(* IEC 61131-3 sources: std_i2980_v2.06_cp053/Source/IMM/ieccontrol/OperationMode1, 14 files *)

(* ---- ABAlarmHandler.pu ---- *)
IMPORT_OVER_LISTFILE
 GET_ALARM_COUNT
, SET_EVENT
, tevAlarmConfirm
, tevPanelButtonRegisterData
, tevPanelButtonRegister
, tsDeviceId
, tevAlarmConfirmData

END_IMPORT

ALGORITHM_BLOCK ABAlarmHandler #DUMMY_EDIT_BLOCK

SYSTEM_VAR
 sv_iPendingAlarms : DINT;
 sv_iPendingMessages : DINT;
 di_ButtonAlarmConfirm : BOOL;
 sv_bLedAlarmConfirm_ledAttr : BYTE (* Panel LED *);
 sv_bLedAlarmConfirm : BOOL;
 sv_bHMILedAlarmConfirm_ledAttr : BYTE (* HMI LED *);
 sv_bHMILedAlarmConfirm : BOOL;
 sv_bAlarmConfirmVis : BOOL;
 sv_bButtonAlarmConfirm : BOOL;
 sv_bInitStart : BOOL;
 sv_DeviceId : tsDeviceId;
END_VAR

SYSTEM_OBJECT
 TaskVis : TASK;
 PU_Task_13 : TASK;
 evAlarmConfirm : tevAlarmConfirm;
 evPanelButtonRegister : tevPanelButtonRegister;
END_OBJECT

VAR
 mAlarmConfirmLedExists : BOOL;
 evPanelButtonRegisterData : tevPanelButtonRegisterData;
 mDIButtonAlarmConfirmLinked : BOOL;
END_VAR

VAR CONSTANT
 cButtonAlarmConfirm : DINT := 5;
END_VAR

POSTUPDATE_ALGORITHM pRegisterButtons ON PU_Task_13 WITH sv_bInitStart

#BEGIN_EDIT_BLOCK

evPanelButtonRegisterData.Button.nPanelButtonType := nPanelButtonAction;
evPanelButtonRegisterData.Button.iCompId := sv_DeviceId.CompId;
evPanelButtonRegisterData.Button.iIndexId := sv_DeviceId.IndexId;
evPanelButtonRegisterData.Button.iButtonId := cButtonAlarmConfirm;
evPanelButtonRegisterData.Button.pbActionVar1 := @sv_bButtonAlarmConfirm;
evPanelButtonRegisterData.Button.Optional.pbLedVar := @sv_bHMILedAlarmConfirm;
evPanelButtonRegisterData.Button.Optional.piLedVarAttr := @sv_bHMILedAlarmConfirm_ledAttr;
SET_EVENT(evPanelButtonRegister, evPanelButtonRegisterData);

mDIButtonAlarmConfirmLinked := IS_LINKED(di_ButtonAlarmConfirm);

;#END_EDIT_BLOCK END_ALGORITHM

PROCESS_ALGORITHM paAlarmCounter ON TaskVis AUTOSTART

VAR
 iChangeCount : DINT;
 iChangeCountOld : DINT;
END_VAR
#BEGIN_EDIT_BLOCK
(**************************************** WARNING ********************************************
 *** The KEBA Kemro K2 System including software is not intended for safety control tasks! ***
 ***                       For further information see Comment tab!                        ***
 *********************************************************************************************)

iChangeCount := GET_ALARM_MODIFICATION_COUNT();
IF iChangeCount <> iChangeCountOld THEN
   sv_iPendingAlarms := (GET_ALARM_COUNT(1)+GET_ALARM_COUNT(2)+GET_ALARM_COUNT(3));
   sv_iPendingMessages := GET_ALARM_COUNT() - sv_iPendingAlarms;
END_IF;
iChangeCountOld := iChangeCount;

;#END_EDIT_BLOCK END_ALGORITHM

POSTUPDATE_ALGORITHM pAlarmConfirmButton ON PU_Task_13 WITH di_ButtonAlarmConfirm,sv_bButtonAlarmConfirm,sv_bAlarmConfirmVis

VAR
 evAlarmConfirmData : tevAlarmConfirmData;
 bButtonAlarmConfirm : BOOL;
END_VAR
#BEGIN_EDIT_BLOCK
(**************************************** WARNING ********************************************
 *** The KEBA Kemro K2 System including software is not intended for safety control tasks! ***
 ***                       For further information see Comment tab!                        ***
 *********************************************************************************************)

bButtonAlarmConfirm := sv_bButtonAlarmConfirm;

IF mDIButtonAlarmConfirmLinked THEN
    bButtonAlarmConfirm := bButtonAlarmConfirm OR di_ButtonAlarmConfirm;
END_IF;

IF (bButtonAlarmConfirm) THEN
    //confirm button on the panel was pressed

    //confirm all alarms
    QUIT_ALARM(Name := ANY,
               SubID1 := ANY,
               SubID2 := ANY,
               SubID3 := ANY,
               SubID4 := ANY);

    //set error confirm event
    evAlarmConfirmData := nConfirmedByPanel;
    SET_EVENT(evAlarmConfirm, evAlarmConfirmData);

ELSIF sv_bAlarmConfirmVis THEN
    //alarms have been confirmed in hmi

    //set error confirm event
    evAlarmConfirmData := nConfirmedByVis;
    SET_EVENT(evAlarmConfirm, evAlarmConfirmData);
    sv_bAlarmConfirmVis := FALSE;
END_IF;

;#END_EDIT_BLOCK END_ALGORITHM

POSTUPDATE_ALGORITHM pLedControl ON PU_Task_13 WITH sv_iPendingAlarms

VAR
 bInitDone : BOOL;
END_VAR
#BEGIN_EDIT_BLOCK
(**************************************** WARNING ********************************************
 *** The KEBA Kemro K2 System including software is not intended for safety control tasks! ***
 ***                       For further information see Comment tab!                        ***
 *********************************************************************************************)

IF NOT bInitDone THEN
    sv_bHMILedAlarmConfirm_ledAttr := 16#1;
    sv_bHMILedAlarmConfirm := FALSE;

    IF (IS_LINKED(sv_bLedAlarmConfirm_ledAttr) AND IS_LINKED(sv_bLedAlarmConfirm)) THEN
        sv_bLedAlarmConfirm_ledAttr := sv_bHMILedAlarmConfirm_ledAttr;
        sv_bLedAlarmConfirm := sv_bHMILedAlarmConfirm;
        mAlarmConfirmLedExists := TRUE;
    ELSE
        mAlarmConfirmLedExists := FALSE;
    END_IF;
    bInitDone := TRUE;
END_IF;

// set the hmi button led
IF sv_iPendingAlarms = 0 THEN
    sv_bHMILedAlarmConfirm := FALSE;
ELSE
    sv_bHMILedAlarmConfirm := TRUE;
END_IF;

IF NOT mAlarmConfirmLedExists THEN
    RETURN;
END_IF;

// set the hw led
IF sv_iPendingAlarms = 0 THEN
    sv_bLedAlarmConfirm := FALSE;
ELSE
    sv_bLedAlarmConfirm := TRUE;
END_IF;

;#END_EDIT_BLOCK END_ALGORITHM

END_ALGORITHM_BLOCK

#END_OF_IEC_PART

@Puma @IecEditor 6 68 @Pou 25
@@@BEG_Comment@@@

@@@END_Comment@@@

@BEG_Contents

@BEG_Func
@RT(17)FuncTreeContainer
2
@Var @RT(15)GET_ALARM_COUNT @RT(0) @T @T @DERIVED 0 @F @RT(22)KEBA_STANDARD_FUNCTION @F
@T
@BEG_Attrib
0 @RT(0) @RT(0)
@END_Attrib
1 1 @F @F @F @F

@Var @RT(9)SET_EVENT @RT(0) @T @T @DERIVED 0 @F @RT(23)KEBA_STANDARD_PROCEDURE @F
@T
@BEG_Attrib
0 @RT(0) @RT(0)
@END_Attrib
1 1 @F @F @F @F

@END_Func

@BEG_Const
@RT(18)ConstTreeContainer
0
@END_Const

@BEG_Export

@BEG_Kind
@ALGORITHM_BLOCK @RT(14)ABAlarmHandler @STRUCTURED_TEXT
@RT(0) @RT(0) @RT(0)
@END_Kind

@BEG_Dcl
@RT(16)DclTreeContainer
19
@Var @RT(7)TaskVis @RT(0) @T @T @RENAMED 0 @T @T @DT @RT(4)TASK @RT(0) @T @T @BASIC 0 @F
@F @F
@T
@BEG_Attrib
3 @RT(0) @RT(0) @RT(0)
@END_Attrib
1 7 @F @F @F @F

@Var @RT(17)sv_iPendingAlarms @RT(0) @T @F @DT @RT(4)DINT @RT(0) @T @T @BASIC 0 @F
@F @F
@T
@BEG_Attrib
3 @RT(0) @RT(0) @RT(0)
@END_Attrib
1 8 @F @F @F @F

@Var @RT(19)sv_iPendingMessages @RT(0) @T @F @DT @RT(4)DINT @RT(0) @T @T @BASIC 0 @F
@F @F
@T
@BEG_Attrib
3 @RT(0) @RT(0) @RT(0)
@END_Attrib
1 8 @F @F @F @F

@Var @RT(21)di_ButtonAlarmConfirm @RT(0) @T @F @DT @RT(4)BOOL @RT(0) @T @T @BASIC 0 @F
@F @F
@T
@BEG_Attrib
3 @RT(0) @RT(0) @RT(0)
@END_Attrib
1 8 @F @F @F @F

@Var @RT(10)PU_Task_13 @RT(0) @T @T @RENAMED 0 @T @T @DT @RT(4)TASK @RT(0) @T @T @BASIC 0 @F
@F @F
@T
@BEG_Attrib
3 @RT(0) @RT(0) @RT(0)
@END_Attrib
1 7 @F @F @F @F

@Var @RT(27)sv_bLedAlarmConfirm_ledAttr @RT(0) @T @F @DT @RT(4)BYTE @RT(0) @T @T @BASIC 0 @F
@F @F
@T
@BEG_Attrib
3 @RT(0) @RT(9)Panel LED @RT(0)
@END_Attrib
1 8 @F @F @F @F

@Var @RT(19)sv_bLedAlarmConfirm @RT(0) @T @F @DT @RT(4)BOOL @RT(0) @T @T @BASIC 0 @F
@F @F
@T
@BEG_Attrib
3 @RT(0) @RT(0) @RT(0)
@END_Attrib
1 8 @F @F @F @F

@Var @RT(30)sv_bHMILedAlarmConfirm_ledAttr @RT(0) @T @F @DT @RT(4)BYTE @RT(0) @T @T @BASIC 0 @F
@F @F
@T
@BEG_Attrib
3 @RT(0) @RT(7)HMI LED @RT(0)
@END_Attrib
1 8 @F @F @F @F

@Var @RT(22)sv_bHMILedAlarmConfirm @RT(0) @T @F @DT @RT(4)BOOL @RT(0) @T @T @BASIC 0 @F
@F @F
@T
@BEG_Attrib
3 @RT(0) @RT(0) @RT(0)
@END_Attrib
1 8 @F @F @F @F

@Var @RT(22)mAlarmConfirmLedExists @RT(0) @T @F @DT @RT(4)BOOL @RT(0) @T @T @BASIC 0 @F
@F @F
@T
@BEG_Attrib
3 @RT(0) @RT(0) @RT(0)
@END_Attrib
1 0 @F @F @F @F

@Var @RT(19)sv_bAlarmConfirmVis @RT(0) @T @T @RENAMED 0 @T @T @DT @RT(4)BOOL @RT(0) @T @T @BASIC 0 @F
@F @F
@T
@BEG_Attrib
3 @RT(0) @RT(0) @RT(0)
@END_Attrib
1 8 @F @F @F @F

@Var @RT(22)sv_bButtonAlarmConfirm @RT(0) @T @F @DT @RT(4)BOOL @RT(0) @T @T @BASIC 0 @F
@F @F
@T
@BEG_Attrib
3 @RT(0) @RT(0) @RT(0)
@END_Attrib
1 8 @F @F @F @F

@Var @RT(14)evAlarmConfirm @RT(0) @T @T @DERIVED 0 @T @T @DT @RT(15)tevAlarmConfirm @RT(0) @T @T @UNKNOWN 0 @F
@F @F
@T
@BEG_Attrib
3 @RT(0) @RT(0) @RT(0)
@END_Attrib
1 7 @F @F @F @F

@Var @RT(25)evPanelButtonRegisterData @RT(0) @T @T @DERIVED 0 @T @T @DT @RT(26)tevPanelButtonRegisterData @RT(0) @T @T @UNKNOWN 0 @F
@F @F
@T
@BEG_Attrib
3 @RT(0) @RT(0) @RT(0)
@END_Attrib
1 0 @F @F @F @F

@Var @RT(21)evPanelButtonRegister @RT(0) @T @T @DERIVED 0 @T @T @DT @RT(22)tevPanelButtonRegister @RT(0) @T @T @UNKNOWN 0 @F
@F @F
@T
@BEG_Attrib
3 @RT(0) @RT(0) @RT(0)
@END_Attrib
1 7 @F @F @F @F

@Var @RT(13)sv_bInitStart @RT(0) @T @T @RENAMED 0 @T @T @DT @RT(4)BOOL @RT(0) @T @T @BASIC 0 @F
@F @F
@T
@BEG_Attrib
3 @RT(0) @RT(0) @RT(0)
@END_Attrib
1 8 @F @F @F @F

@Var @RT(11)sv_DeviceId @RT(0) @T @T @DERIVED 0 @T @T @DT @RT(10)tsDeviceId @RT(0) @T @T @UNKNOWN 0 @F
@F @F
@T
@BEG_Attrib
3 @RT(0) @RT(0) @RT(0)
@END_Attrib
1 8 @F @F @F @F

@Var @RT(27)mDIButtonAlarmConfirmLinked @RT(0) @T @F @DT @RT(4)BOOL @RT(0) @T @T @BASIC 0 @F
@F @F
@T
@BEG_Attrib
3 @RT(0) @RT(0) @RT(0)
@END_Attrib
1 0 @F @F @F @F

@Var @RT(19)cButtonAlarmConfirm @RT(0) @T @F @DT @RT(4)DINT @RT(0) @T @T @BASIC 0 @F
@F @F
@T
@BEG_Attrib
3 @RT(1)5 @RT(0) @RT(0)
@END_Attrib
1 15 @F @F @F @F

@END_Dcl

@END_Export

@BEG_Body

4

@BEG_Export

@BEG_Algo
@POSTUPDATE_ALGORITHM @RT(16)pRegisterButtons @STRUCTURED_TEXT
@RT(0) @RT(13)sv_bInitStart @RT(10)PU_Task_13 @F @F
@END_Algo

@BEG_Dcl
@RT(16)DclTreeContainer
0
@END_Dcl

@END_Export

@BEG_Export

@BEG_Algo
@PROCESS_ALGORITHM @RT(14)paAlarmCounter @STRUCTURED_TEXT
@RT(0) @RT(0) @RT(7)TaskVis @T @F
@END_Algo

@BEG_Dcl
@RT(16)DclTreeContainer
2
@Var @RT(12)iChangeCount @RT(0) @T @F @DT @RT(4)DINT @RT(0) @T @T @BASIC 0 @F
@F @F
@T
@BEG_Attrib
3 @RT(0) @RT(0) @RT(0)
@END_Attrib
1 0 @F @F @F @F

@Var @RT(15)iChangeCountOld @RT(0) @T @F @DT @RT(4)DINT @RT(0) @T @T @BASIC 0 @F
@F @F
@T
@BEG_Attrib
3 @RT(0) @RT(0) @RT(0)
@END_Attrib
1 0 @F @F @F @F

@END_Dcl

@END_Export

@BEG_Export

@BEG_Algo
@POSTUPDATE_ALGORITHM @RT(19)pAlarmConfirmButton @STRUCTURED_TEXT
@RT(0) @RT(64)di_ButtonAlarmConfirm,sv_bButtonAlarmConfirm,sv_bAlarmConfirmVis @RT(10)PU_Task_13 @F @F
@END_Algo

@BEG_Dcl
@RT(16)DclTreeContainer
2
@Var @RT(18)evAlarmConfirmData @RT(0) @T @T @DERIVED 0 @T @T @DT @RT(19)tevAlarmConfirmData @RT(0) @T @T @UNKNOWN 0 @F
@F @F
@T
@BEG_Attrib
3 @RT(0) @RT(0) @RT(0)
@END_Attrib
1 0 @F @F @F @F

@Var @RT(19)bButtonAlarmConfirm @RT(0) @T @F @DT @RT(4)BOOL @RT(0) @T @T @BASIC 0 @F
@F @F
@T
@BEG_Attrib
3 @RT(0) @RT(0) @RT(0)
@END_Attrib
1 0 @F @F @F @F

@END_Dcl

@END_Export

@BEG_Export

@BEG_Algo
@POSTUPDATE_ALGORITHM @RT(11)pLedControl @STRUCTURED_TEXT
@RT(0) @RT(17)sv_iPendingAlarms @RT(10)PU_Task_13 @F @F
@END_Algo

@BEG_Dcl
@RT(16)DclTreeContainer
1
@Var @RT(9)bInitDone @RT(0) @T @F @DT @RT(4)BOOL @RT(0) @T @T @BASIC 0 @F
@F @F
@T
@BEG_Attrib
3 @RT(0) @RT(0) @RT(0)
@END_Attrib
1 0 @F @F @F @F

@END_Dcl

@END_Export

@BEG_Body
@TL(12)

evPanelButtonRegisterData.Button.nPanelButtonType := nPanelButtonAction;
evPanelButtonRegisterData.Button.iCompId := sv_DeviceId.CompId;
evPanelButtonRegisterData.Button.iIndexId := sv_DeviceId.IndexId;
evPanelButtonRegisterData.Button.iButtonId := cButtonAlarmConfirm;
evPanelButtonRegisterData.Button.pbActionVar1 := @sv_bButtonAlarmConfirm;
evPanelButtonRegisterData.Button.Optional.pbLedVar := @sv_bHMILedAlarmConfirm;
evPanelButtonRegisterData.Button.Optional.piLedVarAttr := @sv_bHMILedAlarmConfirm_ledAttr;
SET_EVENT(evPanelButtonRegister, evPanelButtonRegisterData);

mDIButtonAlarmConfirmLinked := IS_LINKED(di_ButtonAlarmConfirm);

@END_Body

@@@BEG_Comment@@@
@TL(0)

@@@END_Comment@@@

@BEG_Body
@TL(15)
(**************************************** WARNING ********************************************
 *** The KEBA Kemro K2 System including software is not intended for safety control tasks! ***
 ***                       For further information see Comment tab!                        ***
 *********************************************************************************************)

iChangeCount := GET_ALARM_MODIFICATION_COUNT();
IF iChangeCount <> iChangeCountOld THEN
   sv_iPendingAlarms := (GET_ALARM_COUNT(1)+GET_ALARM_COUNT(2)+GET_ALARM_COUNT(3));
   sv_iPendingMessages := GET_ALARM_COUNT() - sv_iPendingAlarms;
END_IF;
iChangeCountOld := iChangeCount;

@END_Body

@@@BEG_Comment@@@
@TL(0)

@@@END_Comment@@@

@BEG_Body
@TL(34)
(**************************************** WARNING ********************************************
 *** The KEBA Kemro K2 System including software is not intended for safety control tasks! ***
 ***                       For further information see Comment tab!                        ***
 *********************************************************************************************)

bButtonAlarmConfirm := sv_bButtonAlarmConfirm;

IF mDIButtonAlarmConfirmLinked THEN
    bButtonAlarmConfirm := bButtonAlarmConfirm OR di_ButtonAlarmConfirm;
END_IF;

IF (bButtonAlarmConfirm) THEN
    //confirm button on the panel was pressed

    //confirm all alarms
    QUIT_ALARM(Name := ANY,
               SubID1 := ANY,
               SubID2 := ANY,
               SubID3 := ANY,
               SubID4 := ANY);

    //set error confirm event
    evAlarmConfirmData := nConfirmedByPanel;
    SET_EVENT(evAlarmConfirm, evAlarmConfirmData);

ELSIF sv_bAlarmConfirmVis THEN
    //alarms have been confirmed in hmi

    //set error confirm event
    evAlarmConfirmData := nConfirmedByVis;
    SET_EVENT(evAlarmConfirm, evAlarmConfirmData);
    sv_bAlarmConfirmVis := FALSE;
END_IF;

@END_Body

@@@BEG_Comment@@@
@TL(0)

@@@END_Comment@@@

@BEG_Body
@TL(38)
(**************************************** WARNING ********************************************
 *** The KEBA Kemro K2 System including software is not intended for safety control tasks! ***
 ***                       For further information see Comment tab!                        ***
 *********************************************************************************************)

IF NOT bInitDone THEN
    sv_bHMILedAlarmConfirm_ledAttr := 16#1;
    sv_bHMILedAlarmConfirm := FALSE;

    IF (IS_LINKED(sv_bLedAlarmConfirm_ledAttr) AND IS_LINKED(sv_bLedAlarmConfirm)) THEN
        sv_bLedAlarmConfirm_ledAttr := sv_bHMILedAlarmConfirm_ledAttr;
        sv_bLedAlarmConfirm := sv_bHMILedAlarmConfirm;
        mAlarmConfirmLedExists := TRUE;
    ELSE
        mAlarmConfirmLedExists := FALSE;
    END_IF;
    bInitDone := TRUE;
END_IF;

// set the hmi button led
IF sv_iPendingAlarms = 0 THEN
    sv_bHMILedAlarmConfirm := FALSE;
ELSE
    sv_bHMILedAlarmConfirm := TRUE;
END_IF;

IF NOT mAlarmConfirmLedExists THEN
    RETURN;
END_IF;

// set the hw led
IF sv_iPendingAlarms = 0 THEN
    sv_bLedAlarmConfirm := FALSE;
ELSE
    sv_bLedAlarmConfirm := TRUE;
END_IF;

@END_Body

@@@BEG_Comment@@@
@TL(0)

@@@END_Comment@@@
@END_Body

@END_Contents

(* ---- ABAlarmSignal.pu ---- *)
IMPORT_OVER_LISTFILE
 IS_LINKED
, ABSignalSetReset
, tevAlarmConfirm
, TON
, tevAlarmConfirmData

END_IMPORT

ALGORITHM_BLOCK ABAlarmSignal #DUMMY_EDIT_BLOCK

SYSTEM_VAR
 sv_bAutoCycleRunning : BOOL;
 do_StoppedLamp : BOOL;
 do_RunningLamp : BOOL;
 sv_bInitDone : BOOL;
 do_AlarmLamp : BOOL (* digital output for alarm lamp *);
 do_Buzzer : BOOL (* digital output for buzzer *);
 sv_iSetAlarmSignalCount : DINT (* counter how many alarms requested the alarm signal (incremented with evAlarmLampBlink event; decremented with evAlarmLampReset) *);
 sv_dBuzzerTime : TIME;
 sv_dBuzzerPulseTime : TIME;
END_VAR

SYSTEM_OBJECT
 PU_Task_7 : TASK;
 EV_Task_7 : TASK;
 TaskMid : TASK;
 evAlarmConfirm : tevAlarmConfirm;
END_OBJECT

VAR
 abSignalSetReset : ABSignalSetReset (* this AB counts the alarmevents for set and reset the alarm signals *);
 mbStopBuzzer : BOOL (* stop buzzer *);
END_VAR

POSTUPDATE_ALGORITHM pSetAlarmSignalCount ON PU_Task_7 WITH sv_bInitDone, sv_iSetAlarmSignalCount, sv_bAutoCycleRunning

VAR
 bInitDone : BOOL;
 bAlarmLampLinked : BOOL;
 bRunningLampLinked : BOOL;
 bStoppedLampLinked : BOOL;
 bBuzzerLinked : BOOL;
 iOldCount : DINT;
 iLamp : DINT;
END_VAR
#BEGIN_EDIT_BLOCK
(**************************************** WARNING ********************************************
 *** The KEBA Kemro K2 System including software is not intended for safety control tasks! ***
 ***                       For further information see Comment tab!                        ***
 *********************************************************************************************)

IF NOT bInitDone THEN
    //check if lamp or buzzer is available
    bAlarmLampLinked := IS_LINKED(do_AlarmLamp);
    bRunningLampLinked := IS_LINKED(do_RunningLamp);
    bStoppedLampLinked := IS_LINKED(do_StoppedLamp);
    bBuzzerLinked := IS_LINKED(do_Buzzer);
    bInitDone := TRUE;
END_IF;

//set or reset alarm lamp if available
IF (sv_iSetAlarmSignalCount > 0) THEN
    iLamp := 0; // alarm
ELSIF (sv_bAutoCycleRunning) THEN
    iLamp := 1; // running
ELSE
    iLamp := 2; // stopped
END_IF;

IF bAlarmLampLinked THEN
    do_AlarmLamp := iLamp = 0;
END_IF;

IF bRunningLampLinked THEN
    do_RunningLamp :=  iLamp = 1;
END_IF;

IF bStoppedLampLinked THEN
    do_StoppedLamp := iLamp = 2;
END_IF;

IF (sv_iSetAlarmSignalCount > iOldCount) AND bBuzzerLinked AND sv_dBuzzerTime > T#0ms THEN
   //start buzzer if a new alarm occured
   mbStopBuzzer := FALSE;
   START_PROCESS_ALGORITHM(paBuzzer);
ELSIF sv_iSetAlarmSignalCount = 0 THEN
   mbStopBuzzer := TRUE;
END_IF;

iOldCount := sv_iSetAlarmSignalCount;

;#END_EDIT_BLOCK END_ALGORITHM

PROCESS_ALGORITHM paBuzzer ON TaskMid

VAR
 // dActTime : TIME;
 // bUseMaxTime : BOOL (* Use max buzzer ring time, if time > 0 otherwise no use *);
 fbTimer : TON;
END_VAR

(* IecGraph-Code *)

(* init step *)
INITIAL_STEP S_Init:
END_STEP

(* steps *)
STEP S_OnTime:
AInitTimer (P);
AGenPulses (N);
END_STEP

ACTION AInitTimer: #BEGIN_EDIT_BLOCK
fbTimer(IN := FALSE, PT := sv_dBuzzerPulseTime);
do_Buzzer := TRUE;

;#END_EDIT_BLOCK END_ACTION (*AInitTimer*)
ACTION AGenPulses: #BEGIN_EDIT_BLOCK
fbTimer(IN := TRUE);
IF fbTimer.Q THEN
   do_Buzzer := NOT do_Buzzer;
   fbTimer(IN := FALSE);
END_IF;

;#END_EDIT_BLOCK END_ACTION (*AGenPulses*)
STEP S_Stop:
AStop (P);
END_STEP

ACTION AStop: #BEGIN_EDIT_BLOCK
do_Buzzer := FALSE;
STOP_PROCESS_ALGORITHM();

;#END_EDIT_BLOCK END_ACTION (*AStop*)

(* transitions *)
TRANSITION TStartBuzzer (* Trans1 *) FROM S_Init TO S_OnTime :=  #BEGIN_EDIT_BLOCK
NOT mbStopBuzzer
;#END_EDIT_BLOCK
END_TRANSITION

TRANSITION TOnTimeReached (* Trans2 *) FROM S_OnTime TO S_Stop :=  #BEGIN_EDIT_BLOCK
S_OnTime.T > sv_dBuzzerTime OR mbStopBuzzer
;#END_EDIT_BLOCK
END_TRANSITION

TRANSITION TStart (* Trans9 *) FROM S_Stop TO S_Init :=  #BEGIN_EDIT_BLOCK
TRUE
;#END_EDIT_BLOCK
END_TRANSITION

(* end IecGraph-Code *)
(* sfc-code *)
(* end sfc-code *)

END_ALGORITHM

EVENT_ALGORITHM evaAlarmConfirm ON EV_Task_7 WITH evAlarmConfirm

VAR_INPUT
 evAlarmConfirmData : tevAlarmConfirmData;
END_VAR
#BEGIN_EDIT_BLOCK
(**************************************** WARNING ********************************************
 *** The KEBA Kemro K2 System including software is not intended for safety control tasks! ***
 ***                       For further information see Comment tab!                        ***
 *********************************************************************************************)

//alarms have been confirmed by user -> stop buzzer
mbStopBuzzer := TRUE;

;#END_EDIT_BLOCK END_ALGORITHM

END_ALGORITHM_BLOCK

#END_OF_IEC_PART

@Puma @IecEditor 6 97 @Pou 25
@@@BEG_Comment@@@

@@@END_Comment@@@

@BEG_Contents

@BEG_Func
@RT(17)FuncTreeContainer
1
@Var @RT(9)IS_LINKED @RT(0) @T @T @DERIVED 0 @F @RT(22)KEBA_STANDARD_FUNCTION @F
@T
@BEG_Attrib
0 @RT(0) @RT(0)
@END_Attrib
1 1 @F @F @F @F

@END_Func

@BEG_Const
@RT(18)ConstTreeContainer
0
@END_Const

@BEG_Export

@BEG_Kind
@ALGORITHM_BLOCK @RT(13)ABAlarmSignal @STRUCTURED_TEXT
@RT(0) @RT(0) @RT(0)
@END_Kind

@BEG_Dcl
@RT(16)DclTreeContainer
15
@Var @RT(9)PU_Task_7 @RT(0) @T @T @RENAMED 0 @T @T @DT @RT(4)TASK @RT(0) @T @T @BASIC 0 @F
@F @F
@T
@BEG_Attrib
3 @RT(0) @RT(0) @RT(0)
@END_Attrib
1 7 @F @F @F @F

@Var @RT(20)sv_bAutoCycleRunning @RT(0) @T @F @DT @RT(4)BOOL @RT(0) @T @T @BASIC 0 @F
@F @F
@T
@BEG_Attrib
3 @RT(0) @RT(0) @RT(0)
@END_Attrib
1 8 @F @F @F @F

@Var @RT(14)do_StoppedLamp @RT(0) @T @F @DT @RT(4)BOOL @RT(0) @T @T @BASIC 0 @F
@F @F
@T
@BEG_Attrib
3 @RT(0) @RT(0) @RT(0)
@END_Attrib
1 8 @F @F @F @F

@Var @RT(14)do_RunningLamp @RT(0) @T @F @DT @RT(4)BOOL @RT(0) @T @T @BASIC 0 @F
@F @F
@T
@BEG_Attrib
3 @RT(0) @RT(0) @RT(0)
@END_Attrib
1 8 @F @F @F @F

@Var @RT(9)EV_Task_7 @RT(0) @T @T @RENAMED 0 @T @T @DT @RT(4)TASK @RT(0) @T @T @BASIC 0 @F
@F @F
@T
@BEG_Attrib
3 @RT(0) @RT(0) @RT(0)
@END_Attrib
1 7 @F @F @F @F

@Var @RT(12)sv_bInitDone @RT(0) @T @F @DT @RT(4)BOOL @RT(0) @T @T @BASIC 0 @F
@F @F
@T
@BEG_Attrib
3 @RT(0) @RT(0) @RT(0)
@END_Attrib
1 8 @F @F @F @F

@Var @RT(16)abSignalSetReset @RT(0) @T @T @DERIVED 0 @T @T @DT @RT(16)ABSignalSetReset @RT(0) @T @T @UNKNOWN 0 @F
@F @F
@T
@BEG_Attrib
3 @RT(0) @RT(66)this AB counts the alarmevents for set and reset the alarm signals @RT(0)
@END_Attrib
1 0 @F @F @F @F

@Var @RT(12)do_AlarmLamp @RT(0) @T @F @DT @RT(4)BOOL @RT(0) @T @T @BASIC 0 @F
@F @F
@T
@BEG_Attrib
3 @RT(0) @RT(29)digital output for alarm lamp @RT(0)
@END_Attrib
1 8 @F @F @F @F

@Var @RT(9)do_Buzzer @RT(0) @T @F @DT @RT(4)BOOL @RT(0) @T @T @BASIC 0 @F
@F @F
@T
@BEG_Attrib
3 @RT(0) @RT(25)digital output for buzzer @RT(0)
@END_Attrib
1 8 @F @F @F @F

@Var @RT(7)TaskMid @RT(0) @T @T @RENAMED 0 @T @T @DT @RT(4)TASK @RT(0) @T @T @BASIC 0 @F
@F @F
@T
@BEG_Attrib
3 @RT(0) @RT(0) @RT(0)
@END_Attrib
1 7 @F @F @F @F

@Var @RT(12)mbStopBuzzer @RT(0) @T @F @DT @RT(4)BOOL @RT(0) @T @T @BASIC 0 @F
@F @F
@T
@BEG_Attrib
3 @RT(0) @RT(11)stop buzzer @RT(0)
@END_Attrib
1 0 @F @F @F @F

@Var @RT(14)evAlarmConfirm @RT(0) @T @T @RENAMED 0 @T @T @DT @RT(15)tevAlarmConfirm @RT(0) @T @T @UNKNOWN 0 @F
@F @F
@T
@BEG_Attrib
3 @RT(0) @RT(0) @RT(0)
@END_Attrib
1 7 @F @F @F @F

@Var @RT(23)sv_iSetAlarmSignalCount @RT(0) @T @F @DT @RT(4)DINT @RT(0) @T @T @BASIC 0 @F
@F @F
@T
@BEG_Attrib
3 @RT(0) @RT(127)counter how many alarms requested the alarm signal (incremented with evAlarmLampBlink event; decremented with evAlarmLampReset) @RT(0)
@END_Attrib
1 8 @F @F @F @F

@Var @RT(14)sv_dBuzzerTime @RT(0) @T @F @DT @RT(4)TIME @RT(0) @T @T @BASIC 0 @F
@F @F
@T
@BEG_Attrib
3 @RT(0) @RT(0) @RT(0)
@END_Attrib
1 8 @F @F @F @F

@Var @RT(19)sv_dBuzzerPulseTime @RT(0) @T @F @DT @RT(4)TIME @RT(0) @T @T @BASIC 0 @F
@F @F
@T
@BEG_Attrib
3 @RT(0) @RT(0) @RT(0)
@END_Attrib
1 8 @F @F @F @F

@END_Dcl

@END_Export

@BEG_Body

3

@BEG_Export

@BEG_Algo
@POSTUPDATE_ALGORITHM @RT(20)pSetAlarmSignalCount @STRUCTURED_TEXT
@RT(0) @RT(59)sv_bInitDone, sv_iSetAlarmSignalCount, sv_bAutoCycleRunning @RT(9)PU_Task_7 @F @F
@END_Algo

@BEG_Dcl
@RT(16)DclTreeContainer
7
@Var @RT(9)bInitDone @RT(0) @T @F @DT @RT(4)BOOL @RT(0) @T @T @BASIC 0 @F
@F @F
@T
@BEG_Attrib
3 @RT(0) @RT(0) @RT(0)
@END_Attrib
1 0 @F @F @F @F

@Var @RT(16)bAlarmLampLinked @RT(0) @T @F @DT @RT(4)BOOL @RT(0) @T @T @BASIC 0 @F
@F @F
@T
@BEG_Attrib
3 @RT(0) @RT(0) @RT(0)
@END_Attrib
1 0 @F @F @F @F

@Var @RT(18)bRunningLampLinked @RT(0) @T @F @DT @RT(4)BOOL @RT(0) @T @T @BASIC 0 @F
@F @F
@T
@BEG_Attrib
3 @RT(0) @RT(0) @RT(0)
@END_Attrib
1 0 @F @F @F @F

@Var @RT(18)bStoppedLampLinked @RT(0) @T @F @DT @RT(4)BOOL @RT(0) @T @T @BASIC 0 @F
@F @F
@T
@BEG_Attrib
3 @RT(0) @RT(0) @RT(0)
@END_Attrib
1 0 @F @F @F @F

@Var @RT(13)bBuzzerLinked @RT(0) @T @F @DT @RT(4)BOOL @RT(0) @T @T @BASIC 0 @F
@F @F
@T
@BEG_Attrib
3 @RT(0) @RT(0) @RT(0)
@END_Attrib
1 0 @F @F @F @F

@Var @RT(9)iOldCount @RT(0) @T @F @DT @RT(4)DINT @RT(0) @T @T @BASIC 0 @F
@F @F
@T
@BEG_Attrib
3 @RT(0) @RT(0) @RT(0)
@END_Attrib
1 0 @F @F @F @F

@Var @RT(5)iLamp @RT(0) @T @F @DT @RT(4)DINT @RT(0) @T @T @BASIC 0 @F
@F @F
@T
@BEG_Attrib
3 @RT(0) @RT(0) @RT(0)
@END_Attrib
1 0 @F @F @F @F

@END_Dcl

@END_Export

@BEG_Export

@BEG_Algo
@PROCESS_ALGORITHM @RT(8)paBuzzer @SEQUENTIAL_FLOW_CHART
@RT(0) @RT(0) @RT(7)TaskMid @F @F
@END_Algo

@BEG_Dcl
@RT(16)DclTreeContainer
3
@Var @RT(8)dActTime @RT(0) @T @F @DT @RT(4)TIME @RT(0) @T @T @BASIC 0 @F
@F @T
@T
@BEG_Attrib
3 @RT(0) @RT(0) @RT(0)
@END_Attrib
1 0 @F @F @F @F

@Var @RT(11)bUseMaxTime @RT(0) @T @F @DT @RT(4)BOOL @RT(0) @T @T @BASIC 0 @F
@F @T
@T
@BEG_Attrib
3 @RT(0) @RT(54)Use max buzzer ring time, if time > 0 otherwise no use @RT(0)
@END_Attrib
1 0 @F @F @F @F

@Var @RT(7)fbTimer @RT(0) @T @T @DERIVED 0 @T @T @DT @RT(3)TON @RT(0) @T @T @UNKNOWN 0 @F
@F @F
@T
@BEG_Attrib
3 @RT(0) @RT(0) @RT(0)
@END_Attrib
1 0 @F @F @F @F

@END_Dcl

@END_Export

@BEG_Export

@BEG_Algo
@EVENT_ALGORITHM @RT(15)evaAlarmConfirm @STRUCTURED_TEXT
@RT(0) @RT(14)evAlarmConfirm @RT(9)EV_Task_7 @F @F
@END_Algo

@BEG_Dcl
@RT(16)DclTreeContainer
1
@Var @RT(18)evAlarmConfirmData @RT(0) @T @T @DERIVED 0 @T @T @DT @RT(19)tevAlarmConfirmData @RT(0) @T @T @UNKNOWN 0 @F
@F @F
@T
@BEG_Attrib
3 @RT(0) @RT(0) @RT(0)
@END_Attrib
1 1 @F @F @F @F

@END_Dcl

@END_Export

@BEG_Body
@TL(45)
(**************************************** WARNING ********************************************
 *** The KEBA Kemro K2 System including software is not intended for safety control tasks! ***
 ***                       For further information see Comment tab!                        ***
 *********************************************************************************************)

IF NOT bInitDone THEN
    //check if lamp or buzzer is available
    bAlarmLampLinked := IS_LINKED(do_AlarmLamp);
    bRunningLampLinked := IS_LINKED(do_RunningLamp);
    bStoppedLampLinked := IS_LINKED(do_StoppedLamp);
    bBuzzerLinked := IS_LINKED(do_Buzzer);
    bInitDone := TRUE;
END_IF;

//set or reset alarm lamp if available
IF (sv_iSetAlarmSignalCount > 0) THEN
    iLamp := 0; // alarm
ELSIF (sv_bAutoCycleRunning) THEN
    iLamp := 1; // running
ELSE
    iLamp := 2; // stopped
END_IF;

IF bAlarmLampLinked THEN
    do_AlarmLamp := iLamp = 0;
END_IF;

IF bRunningLampLinked THEN
    do_RunningLamp :=  iLamp = 1;
END_IF;

IF bStoppedLampLinked THEN
    do_StoppedLamp := iLamp = 2;
END_IF;

IF (sv_iSetAlarmSignalCount > iOldCount) AND bBuzzerLinked AND sv_dBuzzerTime > T#0ms THEN
   //start buzzer if a new alarm occured
   mbStopBuzzer := FALSE;
   START_PROCESS_ALGORITHM(paBuzzer);
ELSIF sv_iSetAlarmSignalCount = 0 THEN
   mbStopBuzzer := TRUE;
END_IF;

iOldCount := sv_iSetAlarmSignalCount;

@END_Body

@@@BEG_Comment@@@
@TL(0)

@@@END_Comment@@@

@BEG_SfcBody
10 7 12

@BEG_SfcData 2
@StepSeq @RT(4)sseq @F 1
@Loop @RT(4)loop @F 2
@StepSeq @RT(3)seq @F 5
@Step @RT(6)S_Init @F @T @F @F @RT(0) @F
@AcbCont @RT(7)unnamed @F 0

@Trans @RT(12)TStartBuzzer @F @T @F @F @T @T @TL(2)
NOT mbStopBuzzer

@RT(6)Trans1 @F
@Step @RT(8)S_OnTime @F @F @F @F @RT(0) @F
@AcbCont @RT(7)unnamed @F 2
@Acb @RT(10)AInitTimer @F @T @RT(1)P @RT(0) @F @F @T @TL(3)
fbTimer(IN := FALSE, PT := sv_dBuzzerPulseTime);
do_Buzzer := TRUE;

@F
@Acb @RT(10)AGenPulses @F @T @RT(1)N @RT(0) @F @F @T @TL(6)
fbTimer(IN := TRUE);
IF fbTimer.Q THEN
   do_Buzzer := NOT do_Buzzer;
   fbTimer(IN := FALSE);
END_IF;

@F

@Trans @RT(14)TOnTimeReached @F @T @F @F @T @T @TL(2)
S_OnTime.T > sv_dBuzzerTime OR mbStopBuzzer

@RT(6)Trans2 @F
@Step @RT(6)S_Stop @F @F @F @F @RT(0) @F
@AcbCont @RT(7)unnamed @F 1
@Acb @RT(5)AStop @F @T @RT(1)P @RT(0) @F @F @T @TL(3)
do_Buzzer := FALSE;
STOP_PROCESS_ALGORITHM();

@F

@Trans @RT(6)TStart @F @T @T @T @T @T @TL(2)
TRUE

@RT(6)Trans9 @F

@END_SfcData
@SaActions 0
@SaTrans 0
@SaExits 0
@END_SfcBody

@@@BEG_Comment@@@
@TL(0)

@@@END_Comment@@@

@BEG_Body
@TL(8)
(**************************************** WARNING ********************************************
 *** The KEBA Kemro K2 System including software is not intended for safety control tasks! ***
 ***                       For further information see Comment tab!                        ***
 *********************************************************************************************)

//alarms have been confirmed by user -> stop buzzer
mbStopBuzzer := TRUE;

@END_Body

@@@BEG_Comment@@@
@TL(0)

@@@END_Comment@@@
@END_Body

@END_Contents

(* ---- ABAlarmSignalList.pu ---- *)
IMPORT_OVER_LISTFILE
 SET_ALARM
, tsListStructAlarmSignal
, tsDeviceId
, FBDebugTrace
, tsTraceLevel
, tsElementAlarmSignal
, tsSearchDataAlarmSignal

END_IMPORT

ALGORITHM_BLOCK ABAlarmSignalList #DUMMY_EDIT_BLOCK

SYSTEM_VAR
 sv_DeviceId : tsDeviceId;
 sv_TraceLevel : tsTraceLevel;
END_VAR

SYSTEM_OBJECT
 erListOverflow : ALARM;
END_OBJECT

VAR
 mListStruct : tsListStructAlarmSignal;
 miNextFree : DINT;
 miLowBound : DINT;
 miHighBound : DINT;
 mbInit : BOOL;
 miLastFound : DINT;
 miActElement : DINT;
 fbDebugTrace : FBDebugTrace;
END_VAR

ALGORITHM aInit

#BEGIN_EDIT_BLOCK
miLowBound := GET_LOW_BOUND(mListStruct.List);
miHighBound := GET_HIGH_BOUND(mListStruct.List);
miNextFree := miLowBound;
miLastFound := miLowBound;
miActElement := miLowBound;
mbInit := TRUE;

;#END_EDIT_BLOCK END_ALGORITHM

ALGORITHM aAdd

VAR_INPUT
 Element : tsElementAlarmSignal;
END_VAR
#BEGIN_EDIT_BLOCK
IF NOT mbInit THEN RETURN;; END_IF;

IF miNextFree < miHighBound THEN

    mListStruct.List[miNextFree] := Element;
    mListStruct.Used[miNextFree] := TRUE;
    miNextFree := miNextFree + 1;
ELSE
    //error: List Full
    SET_ALARM(Name := erListOverflow,
              SubID1 := sv_DeviceId.CompId,
              SubID2 := sv_DeviceId.IndexId,
              Param1 := 'ABAlarmSignalList.aAdd');
END_IF;

;#END_EDIT_BLOCK END_ALGORITHM

ALGORITHM aAddAt

VAR_INPUT
 Element : tsElementAlarmSignal;
 iPos : DINT;
END_VAR

VAR_TEMP
 i : DINT;
END_VAR

VAR
 iStart : DINT;
 iEnd : DINT;
END_VAR
#BEGIN_EDIT_BLOCK
IF NOT mbInit THEN RETURN; END_IF;

IF miNextFree <= miHighBound THEN
    IF iPos < miHighBound AND iPos >= miLowBound THEN

        IF iPos < miNextFree THEN

            iStart := miNextFree;
            iEnd := iPos+1;
        ELSE
            i := iPos;
            iEnd := miNextFree;
        END_IF;
        miNextFree := i + 1;

        //reorganize list
        FOR i := iStart TO iEnd BY -1 DO
            mListStruct.List[i] := mListStruct.List[i-1];
            mListStruct.Used[i] := TRUE;
        END_FOR;
        //adding Element
        mListStruct.List[iPos] := Element;
        mListStruct.Used[iPos] := TRUE;
    ELSE
        //error: out of bounds
        IF sv_TraceLevel.bApplication THEN
            fbDebugTrace(sText := 'ABAlarmSignalList.aAddAt: Error: Out of ListBounds');
        END_IF;
    END_IF;
ELSE
    //error: List Full
    SET_ALARM(Name := erListOverflow,
            SubID1 := sv_DeviceId.CompId,
            SubID2 := sv_DeviceId.IndexId,
            Param1 := 'ABAlarmSignalList.aAddAt');
END_IF;

;#END_EDIT_BLOCK END_ALGORITHM

ALGORITHM aSearch

VAR_INPUT
 SearchData : tsSearchDataAlarmSignal;
END_VAR

VAR_OUTPUT
 Element : tsElementAlarmSignal;
 iPos : DINT;
 bFound : BOOL;
END_VAR

VAR_TEMP
 i : DINT;
END_VAR
#BEGIN_EDIT_BLOCK
IF NOT mbInit THEN RETURN;; END_IF;

iPos := 0;
bFound := FALSE;

FOR i := miLowBound TO miNextFree-1 DO

    IF mListStruct.List[i].SearchData = SearchData THEN

       Element := mListStruct.List[i];
       //remember foundposition for aSearchNext
       miLastFound := i;
       iPos := i;
       bFound := TRUE;
       RETURN;;
    END_IF;
END_FOR;

;#END_EDIT_BLOCK END_ALGORITHM

ALGORITHM aSearchNext

VAR_INPUT
 SearchData : tsSearchDataAlarmSignal;
END_VAR

VAR_OUTPUT
 Element : tsElementAlarmSignal;
 iPos : DINT;
 bFound : BOOL;
END_VAR

VAR_TEMP
 i : DINT;
END_VAR
#BEGIN_EDIT_BLOCK
IF NOT mbInit THEN RETURN;; END_IF;

iPos := 0;
bFound := FALSE;

FOR i := miLastFound+1 TO miNextFree-1 DO

    IF mListStruct.List[i].SearchData = SearchData THEN

       Element := mListStruct.List[i];
       //remember foundposition for then next aSearchNext
       miLastFound := i;
       iPos := i;
       bFound := TRUE;
       RETURN;;
    END_IF;
END_FOR;

;#END_EDIT_BLOCK END_ALGORITHM

ALGORITHM aRemove

VAR_INPUT
 SearchData : tsSearchDataAlarmSignal;
END_VAR

VAR_OUTPUT
 Element : tsElementAlarmSignal;
 iPos : DINT;
 bFound : BOOL;
END_VAR

VAR_TEMP
 i : DINT;
END_VAR
#BEGIN_EDIT_BLOCK
IF NOT mbInit THEN RETURN; END_IF;

iPos := 0;
bFound := FALSE;

FOR i := miLowBound TO miNextFree-1 DO

    IF mListStruct.List[i].SearchData = SearchData THEN

       iPos := i;
       bFound := TRUE;
       Element := mListStruct.List[i];
       //reorganize list
       FOR i := iPos TO miNextFree-1 DO
           mListStruct.List[i] := mListStruct.List[i+1];
       END_FOR;
       mListStruct.Used[miNextFree-1] := FALSE;
       miNextFree := miNextFree - 1;
       RETURN;
    END_IF;
END_FOR;

;#END_EDIT_BLOCK END_ALGORITHM

ALGORITHM aRemoveAt

VAR_INPUT
 iPos : DINT;
END_VAR

VAR_OUTPUT
 Element : tsElementAlarmSignal;
END_VAR

VAR_TEMP
 i : DINT;
END_VAR
#BEGIN_EDIT_BLOCK
IF NOT mbInit THEN RETURN; END_IF;

IF iPos <= miHighBound AND iPos >= miLowBound THEN

    Element:= mListStruct.List[iPos];
    miActElement := iPos;

    //reorganize list
    FOR i := iPos TO miNextFree-1 DO
        mListStruct.List[i] := mListStruct.List[i+1];
    END_FOR;
    mListStruct.Used[miNextFree-1] := FALSE;

    miNextFree := miNextFree - 1;
ELSE
    //error: out of bounds
    IF sv_TraceLevel.bApplication THEN
        fbDebugTrace(sText := 'ABAlarmSignalList.aRemoveAt: Error: Out of ListBounds');
    END_IF;
END_IF;

;#END_EDIT_BLOCK END_ALGORITHM

ALGORITHM aRemoveAll

VAR_TEMP
 i : DINT;
END_VAR
#BEGIN_EDIT_BLOCK
IF NOT mbInit THEN RETURN; END_IF;
FOR i := miNextFree-1 TO miLowBound DO
    //clearing the whole list
    mListStruct.Used[i] := FALSE;
END_FOR;
miNextFree := miLowBound;

;#END_EDIT_BLOCK END_ALGORITHM

ALGORITHM aElementAt

VAR_OUTPUT
 Element : tsElementAlarmSignal;
END_VAR

VAR_INPUT
 iPos : DINT;
END_VAR
#BEGIN_EDIT_BLOCK
IF NOT mbInit THEN RETURN; END_IF;

IF iPos <= miHighBound AND iPos >= miLowBound THEN

    Element := mListStruct.List[iPos];
    miActElement := iPos;
ELSE
    //error: out of bounds
    IF sv_TraceLevel.bApplication THEN
        fbDebugTrace(sText := 'ABAlarmSignalList.aElementAt: Error: Out of ListBounds');
    END_IF;
END_IF;

;#END_EDIT_BLOCK END_ALGORITHM

ALGORITHM aModifyAt

VAR_INPUT
 iPos : DINT;
END_VAR

VAR_IN_OUT
 Element : tsElementAlarmSignal;
END_VAR
#BEGIN_EDIT_BLOCK
IF NOT mbInit THEN RETURN; END_IF;

IF iPos <= miHighBound AND iPos >= miLowBound THEN

     mListStruct.List[iPos] := Element;
     miActElement := iPos;
ELSE
    //error: out of bounds
    IF sv_TraceLevel.bApplication THEN
        fbDebugTrace(sText := 'ABAlarmSignalList.aModifyAt: Error: Out of ListBounds');
    END_IF;
END_IF;

;#END_EDIT_BLOCK END_ALGORITHM

// ALGORITHM aGetSize

// #BEGIN_EDIT_BLOCK
// IF NOT mbInit THEN RETURN; END_IF;
// //returns the size of the list
// iSize := miHighBound - miLowBound;

// ;#END_EDIT_BLOCK END_ALGORITHM

// ALGORITHM aGetElementsCount

// VAR_OUTPUT
 // iUsed : DINT;
// END_VAR
// #BEGIN_EDIT_BLOCK
// IF NOT mbInit THEN RETURN; END_IF;
//
// iUsed := miNextFree - miLowBound;

// ;#END_EDIT_BLOCK END_ALGORITHM

FUNCTION aGetSize : DINT
 #DUMMY_EDIT_BLOCK
#BEGIN_EDIT_BLOCK
IF NOT mbInit THEN RETURN; END_IF;
//returns the size of the list
aGetSize := miHighBound - miLowBound;

;#END_EDIT_BLOCK END_FUNCTION

FUNCTION aGetElementCount : DINT
 #DUMMY_EDIT_BLOCK
#BEGIN_EDIT_BLOCK
IF NOT mbInit THEN RETURN; END_IF;

aGetElementCount:= miNextFree - miLowBound;

;#END_EDIT_BLOCK END_FUNCTION

ALGORITHM aFirstElement

VAR_OUTPUT
 Element : tsElementAlarmSignal;
END_VAR
#BEGIN_EDIT_BLOCK
IF NOT mbInit THEN RETURN; END_IF;

miActElement := miLowBound;
Element := mListStruct.List[miLowBound];

;#END_EDIT_BLOCK END_ALGORITHM

ALGORITHM aNextElement

VAR_OUTPUT
 Element : tsElementAlarmSignal;
 iPos : DINT;
END_VAR
#BEGIN_EDIT_BLOCK
IF NOT mbInit THEN RETURN; END_IF;

IF miActElement < miHighBound THEN

    miActElement := miActElement + 1;
    iPos := miActElement;
    Element := mListStruct.List[miActElement];
END_IF;

;#END_EDIT_BLOCK END_ALGORITHM

ALGORITHM aLastElement

VAR_OUTPUT
 Element : tsElementAlarmSignal;
END_VAR
#BEGIN_EDIT_BLOCK
IF NOT mbInit THEN RETURN; END_IF;

miActElement := miNextFree - 1;
Element := mListStruct.List[miActElement];

;#END_EDIT_BLOCK END_ALGORITHM

ALGORITHM aPrevElement

VAR_OUTPUT
 Element : tsElementAlarmSignal;
 iPos : DINT;
END_VAR
#BEGIN_EDIT_BLOCK
IF NOT mbInit THEN RETURN; END_IF;

IF miActElement > miLowBound THEN

    miActElement := miActElement - 1;
    iPos := miActElement;
    Element := mListStruct.List[miActElement];
END_IF;

;#END_EDIT_BLOCK END_ALGORITHM

ALGORITHM aImport

VAR_INPUT
 ListStruct : tsListStructAlarmSignal;
END_VAR

VAR_TEMP
 i : DINT;
END_VAR
#BEGIN_EDIT_BLOCK
IF NOT mbInit THEN RETURN; END_IF;

miLastFound := miLowBound;
miActElement := miLowBound;
miNextFree := miLowBound;
mListStruct :=  ListStruct;

//cheching used elements
FOR i := miLowBound TO miHighBound DO

   IF NOT mListStruct.Used[i] THEN
        miNextFree := i;
        RETURN;
   END_IF;
END_FOR;

;#END_EDIT_BLOCK END_ALGORITHM

ALGORITHM aExport

VAR_OUTPUT
 ListStruct : tsListStructAlarmSignal;
END_VAR
#BEGIN_EDIT_BLOCK
IF NOT mbInit THEN RETURN; END_IF;

ListStruct := mListStruct;

;#END_EDIT_BLOCK END_ALGORITHM

END_ALGORITHM_BLOCK

#END_OF_IEC_PART

@Puma @IecEditor 6 68 @Pou 25
@@@BEG_Comment@@@

@@@END_Comment@@@

@BEG_Contents

@BEG_Func
@RT(17)FuncTreeContainer
1
@Var @RT(9)SET_ALARM @RT(0) @T @T @DERIVED 0 @F @RT(23)KEBA_STANDARD_PROCEDURE @F
@T
@BEG_Attrib
0 @RT(0) @RT(0)
@END_Attrib
1 1 @F @F @F @F

@END_Func

@BEG_Const
@RT(18)ConstTreeContainer
0
@END_Const

@BEG_Export

@BEG_Kind
@ALGORITHM_BLOCK @RT(17)ABAlarmSignalList @STRUCTURED_TEXT
@RT(0) @RT(0) @RT(0)
@END_Kind

@BEG_Dcl
@RT(16)DclTreeContainer
11
@Var @RT(14)erListOverflow @RT(0) @T @F @DT @RT(5)ALARM @RT(0) @T @T @BASIC 0 @F
@F @F
@T
@BEG_Attrib
3 @RT(0) @RT(0) @RT(0)
@END_Attrib
1 7 @F @F @F @F

@Var @RT(11)mListStruct @RT(0) @T @T @DERIVED 0 @T @T @DT @RT(23)tsListStructAlarmSignal @RT(0) @T @T @UNKNOWN 0 @F
@F @F
@T
@BEG_Attrib
3 @RT(0) @RT(0) @RT(0)
@END_Attrib
1 0 @F @F @F @F

@Var @RT(10)miNextFree @RT(0) @T @F @DT @RT(4)DINT @RT(0) @T @T @BASIC 0 @F
@F @F
@T
@BEG_Attrib
3 @RT(0) @RT(0) @RT(0)
@END_Attrib
1 0 @F @F @F @F

@Var @RT(10)miLowBound @RT(0) @T @F @DT @RT(4)DINT @RT(0) @T @T @BASIC 0 @F
@F @F
@T
@BEG_Attrib
3 @RT(0) @RT(0) @RT(0)
@END_Attrib
1 0 @F @F @F @F

@Var @RT(11)miHighBound @RT(0) @T @F @DT @RT(4)DINT @RT(0) @T @T @BASIC 0 @F
@F @F
@T
@BEG_Attrib
3 @RT(0) @RT(0) @RT(0)
@END_Attrib
1 0 @F @F @F @F

@Var @RT(6)mbInit @RT(0) @T @F @DT @RT(4)BOOL @RT(0) @T @T @BASIC 0 @F
@F @F
@T
@BEG_Attrib
3 @RT(0) @RT(0) @RT(0)
@END_Attrib
1 0 @F @F @F @F

@Var @RT(11)miLastFound @RT(0) @T @F @DT @RT(4)DINT @RT(0) @T @T @BASIC 0 @F
@F @F
@T
@BEG_Attrib
3 @RT(0) @RT(0) @RT(0)
@END_Attrib
1 0 @F @F @F @F

@Var @RT(12)miActElement @RT(0) @T @F @DT @RT(4)DINT @RT(0) @T @T @BASIC 0 @F
@F @F
@T
@BEG_Attrib
3 @RT(0) @RT(0) @RT(0)
@END_Attrib
1 0 @F @F @F @F

@Var @RT(11)sv_DeviceId @RT(0) @T @T @DERIVED 0 @T @T @DT @RT(10)tsDeviceId @RT(0) @T @T @UNKNOWN 0 @F
@F @F
@T
@BEG_Attrib
3 @RT(0) @RT(0) @RT(0)
@END_Attrib
1 8 @F @F @F @F

@Var @RT(12)fbDebugTrace @RT(0) @T @T @DERIVED 0 @T @T @DT @RT(12)FBDebugTrace @RT(0) @T @T @UNKNOWN 0 @F
@F @F
@T
@BEG_Attrib
3 @RT(0) @RT(0) @RT(0)
@END_Attrib
1 0 @F @F @F @F

@Var @RT(13)sv_TraceLevel @RT(0) @T @T @DERIVED 0 @T @T @DT @RT(12)tsTraceLevel @RT(0) @T @T @UNKNOWN 0 @F
@F @F
@T
@BEG_Attrib
3 @RT(0) @RT(0) @RT(0)
@END_Attrib
1 8 @F @F @F @F

@END_Dcl

@END_Export

@BEG_Body

20

@BEG_Export

@BEG_Algo
@ALGORITHM @RT(5)aInit @STRUCTURED_TEXT
@RT(0) @RT(0) @RT(0) @F @F
@END_Algo

@BEG_Dcl
@RT(16)DclTreeContainer
0
@END_Dcl

@END_Export

@BEG_Export

@BEG_Algo
@ALGORITHM @RT(4)aAdd @STRUCTURED_TEXT
@RT(0) @RT(0) @RT(0) @F @F
@END_Algo

@BEG_Dcl
@RT(16)DclTreeContainer
1
@Var @RT(7)Element @RT(0) @T @T @DERIVED 0 @T @T @DT @RT(20)tsElementAlarmSignal @RT(0) @T @T @UNKNOWN 0 @F
@F @F
@T
@BEG_Attrib
3 @RT(0) @RT(0) @RT(0)
@END_Attrib
1 1 @F @F @F @F

@END_Dcl

@END_Export

@BEG_Export

@BEG_Algo
@ALGORITHM @RT(6)aAddAt @STRUCTURED_TEXT
@RT(0) @RT(0) @RT(0) @F @F
@END_Algo

@BEG_Dcl
@RT(16)DclTreeContainer
5
@Var @RT(7)Element @RT(0) @T @T @DERIVED 0 @T @T @DT @RT(20)tsElementAlarmSignal @RT(0) @T @T @UNKNOWN 0 @F
@F @F
@T
@BEG_Attrib
3 @RT(0) @RT(0) @RT(0)
@END_Attrib
1 1 @F @F @F @F

@Var @RT(4)iPos @RT(0) @T @F @DT @RT(4)DINT @RT(0) @T @T @BASIC 0 @F
@F @F
@T
@BEG_Attrib
3 @RT(0) @RT(0) @RT(0)
@END_Attrib
1 1 @F @F @F @F

@Var @RT(1)i @RT(0) @T @F @DT @RT(4)DINT @RT(0) @T @T @BASIC 0 @F
@F @F
@T
@BEG_Attrib
3 @RT(0) @RT(0) @RT(0)
@END_Attrib
1 4 @F @F @F @F

@Var @RT(6)iStart @RT(0) @T @F @DT @RT(4)DINT @RT(0) @T @T @BASIC 0 @F
@F @F
@T
@BEG_Attrib
3 @RT(0) @RT(0) @RT(0)
@END_Attrib
1 0 @F @F @F @F

@Var @RT(4)iEnd @RT(0) @T @F @DT @RT(4)DINT @RT(0) @T @T @BASIC 0 @F
@F @F
@T
@BEG_Attrib
3 @RT(0) @RT(0) @RT(0)
@END_Attrib
1 0 @F @F @F @F

@END_Dcl

@END_Export

@BEG_Export

@BEG_Algo
@ALGORITHM @RT(7)aSearch @STRUCTURED_TEXT
@RT(0) @RT(0) @RT(0) @F @F
@END_Algo

@BEG_Dcl
@RT(16)DclTreeContainer
5
@Var @RT(10)SearchData @RT(0) @T @T @DERIVED 0 @T @T @DT @RT(23)tsSearchDataAlarmSignal @RT(0) @T @T @UNKNOWN 0 @F
@F @F
@T
@BEG_Attrib
3 @RT(0) @RT(0) @RT(0)
@END_Attrib
1 1 @F @F @F @F

@Var @RT(7)Element @RT(0) @T @T @DERIVED 0 @T @T @DT @RT(20)tsElementAlarmSignal @RT(0) @T @T @UNKNOWN 0 @F
@F @F
@T
@BEG_Attrib
3 @RT(0) @RT(0) @RT(0)
@END_Attrib
1 3 @F @F @F @F

@Var @RT(4)iPos @RT(0) @T @F @DT @RT(4)DINT @RT(0) @T @T @BASIC 0 @F
@F @F
@T
@BEG_Attrib
3 @RT(0) @RT(0) @RT(0)
@END_Attrib
1 3 @F @F @F @F

@Var @RT(6)bFound @RT(0) @T @F @DT @RT(4)BOOL @RT(0) @T @T @BASIC 0 @F
@F @F
@T
@BEG_Attrib
3 @RT(0) @RT(0) @RT(0)
@END_Attrib
1 3 @F @F @F @F

@Var @RT(1)i @RT(0) @T @F @DT @RT(4)DINT @RT(0) @T @T @BASIC 0 @F
@F @F
@T
@BEG_Attrib
3 @RT(0) @RT(0) @RT(0)
@END_Attrib
1 4 @F @F @F @F

@END_Dcl

@END_Export

@BEG_Export

@BEG_Algo
@ALGORITHM @RT(11)aSearchNext @STRUCTURED_TEXT
@RT(0) @RT(0) @RT(0) @F @F
@END_Algo

@BEG_Dcl
@RT(16)DclTreeContainer
5
@Var @RT(10)SearchData @RT(0) @T @T @DERIVED 0 @T @T @DT @RT(23)tsSearchDataAlarmSignal @RT(0) @T @T @UNKNOWN 0 @F
@F @F
@T
@BEG_Attrib
3 @RT(0) @RT(0) @RT(0)
@END_Attrib
1 1 @F @F @F @F

@Var @RT(7)Element @RT(0) @T @T @DERIVED 0 @T @T @DT @RT(20)tsElementAlarmSignal @RT(0) @T @T @UNKNOWN 0 @F
@F @F
@T
@BEG_Attrib
3 @RT(0) @RT(0) @RT(0)
@END_Attrib
1 3 @F @F @F @F

@Var @RT(4)iPos @RT(0) @T @F @DT @RT(4)DINT @RT(0) @T @T @BASIC 0 @F
@F @F
@T
@BEG_Attrib
3 @RT(0) @RT(0) @RT(0)
@END_Attrib
1 3 @F @F @F @F

@Var @RT(6)bFound @RT(0) @T @F @DT @RT(4)BOOL @RT(0) @T @T @BASIC 0 @F
@F @F
@T
@BEG_Attrib
3 @RT(0) @RT(0) @RT(0)
@END_Attrib
1 3 @F @F @F @F

@Var @RT(1)i @RT(0) @T @F @DT @RT(4)DINT @RT(0) @T @T @BASIC 0 @F
@F @F
@T
@BEG_Attrib
3 @RT(0) @RT(0) @RT(0)
@END_Attrib
1 4 @F @F @F @F

@END_Dcl

@END_Export

@BEG_Export

@BEG_Algo
@ALGORITHM @RT(7)aRemove @STRUCTURED_TEXT
@RT(0) @RT(0) @RT(0) @F @F
@END_Algo

@BEG_Dcl
@RT(16)DclTreeContainer
5
@Var @RT(10)SearchData @RT(0) @T @T @DERIVED 0 @T @T @DT @RT(23)tsSearchDataAlarmSignal @RT(0) @T @T @UNKNOWN 0 @F
@F @F
@T
@BEG_Attrib
3 @RT(0) @RT(0) @RT(0)
@END_Attrib
1 1 @F @F @F @F

@Var @RT(7)Element @RT(0) @T @T @DERIVED 0 @T @T @DT @RT(20)tsElementAlarmSignal @RT(0) @T @T @UNKNOWN 0 @F
@F @F
@T
@BEG_Attrib
3 @RT(0) @RT(0) @RT(0)
@END_Attrib
1 3 @F @F @F @F

@Var @RT(4)iPos @RT(0) @T @F @DT @RT(4)DINT @RT(0) @T @T @BASIC 0 @F
@F @F
@T
@BEG_Attrib
3 @RT(0) @RT(0) @RT(0)
@END_Attrib
1 3 @F @F @F @F

@Var @RT(6)bFound @RT(0) @T @F @DT @RT(4)BOOL @RT(0) @T @T @BASIC 0 @F
@F @F
@T
@BEG_Attrib
3 @RT(0) @RT(0) @RT(0)
@END_Attrib
1 3 @F @F @F @F

@Var @RT(1)i @RT(0) @T @F @DT @RT(4)DINT @RT(0) @T @T @BASIC 0 @F
@F @F
@T
@BEG_Attrib
3 @RT(0) @RT(0) @RT(0)
@END_Attrib
1 4 @F @F @F @F

@END_Dcl

@END_Export

@BEG_Export

@BEG_Algo
@ALGORITHM @RT(9)aRemoveAt @STRUCTURED_TEXT
@RT(0) @RT(0) @RT(0) @F @F
@END_Algo

@BEG_Dcl
@RT(16)DclTreeContainer
3
@Var @RT(4)iPos @RT(0) @T @F @DT @RT(4)DINT @RT(0) @T @T @BASIC 0 @F
@F @F
@T
@BEG_Attrib
3 @RT(0) @RT(0) @RT(0)
@END_Attrib
1 1 @F @F @F @F

@Var @RT(7)Element @RT(0) @T @T @DERIVED 0 @T @T @DT @RT(20)tsElementAlarmSignal @RT(0) @T @T @UNKNOWN 0 @F
@F @F
@T
@BEG_Attrib
3 @RT(0) @RT(0) @RT(0)
@END_Attrib
1 3 @F @F @F @F

@Var @RT(1)i @RT(0) @T @F @DT @RT(4)DINT @RT(0) @T @T @BASIC 0 @F
@F @F
@T
@BEG_Attrib
3 @RT(0) @RT(0) @RT(0)
@END_Attrib
1 4 @F @F @F @F

@END_Dcl

@END_Export

@BEG_Export

@BEG_Algo
@ALGORITHM @RT(10)aRemoveAll @STRUCTURED_TEXT
@RT(0) @RT(0) @RT(0) @F @F
@END_Algo

@BEG_Dcl
@RT(16)DclTreeContainer
1
@Var @RT(1)i @RT(0) @T @F @DT @RT(4)DINT @RT(0) @T @T @BASIC 0 @F
@F @F
@T
@BEG_Attrib
3 @RT(0) @RT(0) @RT(0)
@END_Attrib
1 4 @F @F @F @F

@END_Dcl

@END_Export

@BEG_Export

@BEG_Algo
@ALGORITHM @RT(10)aElementAt @STRUCTURED_TEXT
@RT(0) @RT(0) @RT(0) @F @F
@END_Algo

@BEG_Dcl
@RT(16)DclTreeContainer
2
@Var @RT(7)Element @RT(0) @T @T @DERIVED 0 @T @T @DT @RT(20)tsElementAlarmSignal @RT(0) @T @T @UNKNOWN 0 @F
@F @F
@T
@BEG_Attrib
3 @RT(0) @RT(0) @RT(0)
@END_Attrib
1 3 @F @F @F @F

@Var @RT(4)iPos @RT(0) @T @F @DT @RT(4)DINT @RT(0) @T @T @BASIC 0 @F
@F @F
@T
@BEG_Attrib
3 @RT(0) @RT(0) @RT(0)
@END_Attrib
1 1 @F @F @F @F

@END_Dcl

@END_Export

@BEG_Export

@BEG_Algo
@ALGORITHM @RT(9)aModifyAt @STRUCTURED_TEXT
@RT(0) @RT(0) @RT(0) @F @F
@END_Algo

@BEG_Dcl
@RT(16)DclTreeContainer
2
@Var @RT(4)iPos @RT(0) @T @F @DT @RT(4)DINT @RT(0) @T @T @BASIC 0 @F
@F @F
@T
@BEG_Attrib
3 @RT(0) @RT(0) @RT(0)
@END_Attrib
1 1 @F @F @F @F

@Var @RT(7)Element @RT(0) @T @T @DERIVED 0 @T @T @DT @RT(20)tsElementAlarmSignal @RT(0) @T @T @UNKNOWN 0 @F
@F @F
@T
@BEG_Attrib
3 @RT(0) @RT(0) @RT(0)
@END_Attrib
1 2 @F @F @F @F

@END_Dcl

@END_Export

@BEG_Export

@BEG_Algo
@ALGORITHM @RT(8)aGetSize @STRUCTURED_TEXT
@RT(0) @RT(0) @RT(0) @F @T
@END_Algo

@BEG_Dcl
@RT(16)DclTreeContainer
0
@END_Dcl

@END_Export

@BEG_Export

@BEG_Algo
@ALGORITHM @RT(17)aGetElementsCount @STRUCTURED_TEXT
@RT(0) @RT(0) @RT(0) @F @T
@END_Algo

@BEG_Dcl
@RT(16)DclTreeContainer
1
@Var @RT(5)iUsed @RT(0) @T @F @DT @RT(4)DINT @RT(0) @T @T @BASIC 0 @F
@F @F
@T
@BEG_Attrib
3 @RT(0) @RT(0) @RT(0)
@END_Attrib
1 3 @F @F @F @F

@END_Dcl

@END_Export

@BEG_Export

@BEG_Algo
@FUNCTION @RT(8)aGetSize @STRUCTURED_TEXT
@RT(4)DINT @RT(0) @RT(0) @F @F
@END_Algo

@BEG_Dcl
@RT(16)DclTreeContainer
0
@END_Dcl

@END_Export

@BEG_Export

@BEG_Algo
@FUNCTION @RT(16)aGetElementCount @STRUCTURED_TEXT
@RT(4)DINT @RT(0) @RT(0) @F @F
@END_Algo

@BEG_Dcl
@RT(16)DclTreeContainer
0
@END_Dcl

@END_Export

@BEG_Export

@BEG_Algo
@ALGORITHM @RT(13)aFirstElement @STRUCTURED_TEXT
@RT(0) @RT(0) @RT(0) @F @F
@END_Algo

@BEG_Dcl
@RT(16)DclTreeContainer
1
@Var @RT(7)Element @RT(0) @T @T @DERIVED 0 @T @T @DT @RT(20)tsElementAlarmSignal @RT(0) @T @T @UNKNOWN 0 @F
@F @F
@T
@BEG_Attrib
3 @RT(0) @RT(0) @RT(0)
@END_Attrib
1 3 @F @F @F @F

@END_Dcl

@END_Export

@BEG_Export

@BEG_Algo
@ALGORITHM @RT(12)aNextElement @STRUCTURED_TEXT
@RT(0) @RT(0) @RT(0) @F @F
@END_Algo

@BEG_Dcl
@RT(16)DclTreeContainer
2
@Var @RT(7)Element @RT(0) @T @T @DERIVED 0 @T @T @DT @RT(20)tsElementAlarmSignal @RT(0) @T @T @UNKNOWN 0 @F
@F @F
@T
@BEG_Attrib
3 @RT(0) @RT(0) @RT(0)
@END_Attrib
1 3 @F @F @F @F

@Var @RT(4)iPos @RT(0) @T @F @DT @RT(4)DINT @RT(0) @T @T @BASIC 0 @F
@F @F
@T
@BEG_Attrib
3 @RT(0) @RT(0) @RT(0)
@END_Attrib
1 3 @F @F @F @F

@END_Dcl

@END_Export

@BEG_Export

@BEG_Algo
@ALGORITHM @RT(12)aLastElement @STRUCTURED_TEXT
@RT(0) @RT(0) @RT(0) @F @F
@END_Algo

@BEG_Dcl
@RT(16)DclTreeContainer
1
@Var @RT(7)Element @RT(0) @T @T @DERIVED 0 @T @T @DT @RT(20)tsElementAlarmSignal @RT(0) @T @T @UNKNOWN 0 @F
@F @F
@T
@BEG_Attrib
3 @RT(0) @RT(0) @RT(0)
@END_Attrib
1 3 @F @F @F @F

@END_Dcl

@END_Export

@BEG_Export

@BEG_Algo
@ALGORITHM @RT(12)aPrevElement @STRUCTURED_TEXT
@RT(0) @RT(0) @RT(0) @F @F
@END_Algo

@BEG_Dcl
@RT(16)DclTreeContainer
2
@Var @RT(7)Element @RT(0) @T @T @DERIVED 0 @T @T @DT @RT(20)tsElementAlarmSignal @RT(0) @T @T @UNKNOWN 0 @F
@F @F
@T
@BEG_Attrib
3 @RT(0) @RT(0) @RT(0)
@END_Attrib
1 3 @F @F @F @F

@Var @RT(4)iPos @RT(0) @T @F @DT @RT(4)DINT @RT(0) @T @T @BASIC 0 @F
@F @F
@T
@BEG_Attrib
3 @RT(0) @RT(0) @RT(0)
@END_Attrib
1 3 @F @F @F @F

@END_Dcl

@END_Export

@BEG_Export

@BEG_Algo
@ALGORITHM @RT(7)aImport @STRUCTURED_TEXT
@RT(0) @RT(0) @RT(0) @F @F
@END_Algo

@BEG_Dcl
@RT(16)DclTreeContainer
2
@Var @RT(10)ListStruct @RT(0) @T @T @DERIVED 0 @T @T @DT @RT(23)tsListStructAlarmSignal @RT(0) @T @T @UNKNOWN 0 @F
@F @F
@T
@BEG_Attrib
3 @RT(0) @RT(0) @RT(0)
@END_Attrib
1 1 @F @F @F @F

@Var @RT(1)i @RT(0) @T @F @DT @RT(4)DINT @RT(0) @T @T @BASIC 0 @F
@F @F
@T
@BEG_Attrib
3 @RT(0) @RT(0) @RT(0)
@END_Attrib
1 4 @F @F @F @F

@END_Dcl

@END_Export

@BEG_Export

@BEG_Algo
@ALGORITHM @RT(7)aExport @STRUCTURED_TEXT
@RT(0) @RT(0) @RT(0) @F @F
@END_Algo

@BEG_Dcl
@RT(16)DclTreeContainer
1
@Var @RT(10)ListStruct @RT(0) @T @T @DERIVED 0 @T @T @DT @RT(23)tsListStructAlarmSignal @RT(0) @T @T @UNKNOWN 0 @F
@F @F
@T
@BEG_Attrib
3 @RT(0) @RT(0) @RT(0)
@END_Attrib
1 3 @F @F @F @F

@END_Dcl

@END_Export

@BEG_Body
@TL(7)
miLowBound := GET_LOW_BOUND(mListStruct.List);
miHighBound := GET_HIGH_BOUND(mListStruct.List);
miNextFree := miLowBound;
miLastFound := miLowBound;
miActElement := miLowBound;
mbInit := TRUE;

@END_Body

@@@BEG_Comment@@@
@TL(0)

@@@END_Comment@@@

@BEG_Body
@TL(15)
IF NOT mbInit THEN RETURN;; END_IF;

IF miNextFree < miHighBound THEN

    mListStruct.List[miNextFree] := Element;
    mListStruct.Used[miNextFree] := TRUE;
    miNextFree := miNextFree + 1;
ELSE
    //error: List Full
    SET_ALARM(Name := erListOverflow,
              SubID1 := sv_DeviceId.CompId,
              SubID2 := sv_DeviceId.IndexId,
              Param1 := 'ABAlarmSignalList.aAdd');
END_IF;

@END_Body

@@@BEG_Comment@@@
@TL(0)

@@@END_Comment@@@

@BEG_Body
@TL(37)
IF NOT mbInit THEN RETURN; END_IF;

IF miNextFree <= miHighBound THEN
    IF iPos < miHighBound AND iPos >= miLowBound THEN

        IF iPos < miNextFree THEN

            iStart := miNextFree;
            iEnd := iPos+1;
        ELSE
            i := iPos;
            iEnd := miNextFree;
        END_IF;
        miNextFree := i + 1;

        //reorganize list
        FOR i := iStart TO iEnd BY -1 DO
            mListStruct.List[i] := mListStruct.List[i-1];
            mListStruct.Used[i] := TRUE;
        END_FOR;
        //adding Element
        mListStruct.List[iPos] := Element;
        mListStruct.Used[iPos] := TRUE;
    ELSE
        //error: out of bounds
        IF sv_TraceLevel.bApplication THEN
            fbDebugTrace(sText := 'ABAlarmSignalList.aAddAt: Error: Out of ListBounds');
        END_IF;
    END_IF;
ELSE
    //error: List Full
    SET_ALARM(Name := erListOverflow,
            SubID1 := sv_DeviceId.CompId,
            SubID2 := sv_DeviceId.IndexId,
            Param1 := 'ABAlarmSignalList.aAddAt');
END_IF;

@END_Body

@@@BEG_Comment@@@
@TL(0)

@@@END_Comment@@@

@BEG_Body
@TL(18)
IF NOT mbInit THEN RETURN;; END_IF;

iPos := 0;
bFound := FALSE;

FOR i := miLowBound TO miNextFree-1 DO

    IF mListStruct.List[i].SearchData = SearchData THEN

       Element := mListStruct.List[i];
       //remember foundposition for aSearchNext
       miLastFound := i;
       iPos := i;
       bFound := TRUE;
       RETURN;;
    END_IF;
END_FOR;

@END_Body

@@@BEG_Comment@@@
@TL(0)

@@@END_Comment@@@

@BEG_Body
@TL(19)
IF NOT mbInit THEN RETURN;; END_IF;

iPos := 0;
bFound := FALSE;

FOR i := miLastFound+1 TO miNextFree-1 DO

    IF mListStruct.List[i].SearchData = SearchData THEN

       Element := mListStruct.List[i];
       //remember foundposition for then next aSearchNext
       miLastFound := i;
       iPos := i;
       bFound := TRUE;
       RETURN;;
    END_IF;
END_FOR;

@END_Body

@@@BEG_Comment@@@
@TL(0)

@@@END_Comment@@@

@BEG_Body
@TL(22)
IF NOT mbInit THEN RETURN; END_IF;

iPos := 0;
bFound := FALSE;

FOR i := miLowBound TO miNextFree-1 DO

    IF mListStruct.List[i].SearchData = SearchData THEN

       iPos := i;
       bFound := TRUE;
       Element := mListStruct.List[i];
       //reorganize list
       FOR i := iPos TO miNextFree-1 DO
           mListStruct.List[i] := mListStruct.List[i+1];
       END_FOR;
       mListStruct.Used[miNextFree-1] := FALSE;
       miNextFree := miNextFree - 1;
       RETURN;
    END_IF;
END_FOR;

@END_Body

@@@BEG_Comment@@@
@TL(0)

@@@END_Comment@@@

@BEG_Body
@TL(21)
IF NOT mbInit THEN RETURN; END_IF;

IF iPos <= miHighBound AND iPos >= miLowBound THEN

    Element:= mListStruct.List[iPos];
    miActElement := iPos;

    //reorganize list
    FOR i := iPos TO miNextFree-1 DO
        mListStruct.List[i] := mListStruct.List[i+1];
    END_FOR;
    mListStruct.Used[miNextFree-1] := FALSE;

    miNextFree := miNextFree - 1;
ELSE
    //error: out of bounds
    IF sv_TraceLevel.bApplication THEN
        fbDebugTrace(sText := 'ABAlarmSignalList.aRemoveAt: Error: Out of ListBounds');
    END_IF;
END_IF;

@END_Body

@@@BEG_Comment@@@
@TL(0)

@@@END_Comment@@@

@BEG_Body
@TL(7)
IF NOT mbInit THEN RETURN; END_IF;
FOR i := miNextFree-1 TO miLowBound DO
    //clearing the whole list
    mListStruct.Used[i] := FALSE;
END_FOR;
miNextFree := miLowBound;

@END_Body

@@@BEG_Comment@@@
@TL(0)

@@@END_Comment@@@

@BEG_Body
@TL(13)
IF NOT mbInit THEN RETURN; END_IF;

IF iPos <= miHighBound AND iPos >= miLowBound THEN

    Element := mListStruct.List[iPos];
    miActElement := iPos;
ELSE
    //error: out of bounds
    IF sv_TraceLevel.bApplication THEN
        fbDebugTrace(sText := 'ABAlarmSignalList.aElementAt: Error: Out of ListBounds');
    END_IF;
END_IF;

@END_Body

@@@BEG_Comment@@@
@TL(0)

@@@END_Comment@@@

@BEG_Body
@TL(13)
IF NOT mbInit THEN RETURN; END_IF;

IF iPos <= miHighBound AND iPos >= miLowBound THEN

     mListStruct.List[iPos] := Element;
     miActElement := iPos;
ELSE
    //error: out of bounds
    IF sv_TraceLevel.bApplication THEN
        fbDebugTrace(sText := 'ABAlarmSignalList.aModifyAt: Error: Out of ListBounds');
    END_IF;
END_IF;

@END_Body

@@@BEG_Comment@@@
@TL(0)

@@@END_Comment@@@

@BEG_Body
@TL(4)
IF NOT mbInit THEN RETURN; END_IF;
//returns the size of the list
iSize := miHighBound - miLowBound;

@END_Body

@@@BEG_Comment@@@
@TL(0)

@@@END_Comment@@@

@BEG_Body
@TL(4)
IF NOT mbInit THEN RETURN; END_IF;

iUsed := miNextFree - miLowBound;

@END_Body

@@@BEG_Comment@@@
@TL(0)

@@@END_Comment@@@

@BEG_Body
@TL(5)
IF NOT mbInit THEN RETURN; END_IF;
//returns the size of the list
aGetSize := miHighBound - miLowBound;

@END_Body

@@@BEG_Comment@@@
@TL(0)

@@@END_Comment@@@

@BEG_Body
@TL(5)
IF NOT mbInit THEN RETURN; END_IF;

aGetElementCount:= miNextFree - miLowBound;

@END_Body

@@@BEG_Comment@@@
@TL(0)

@@@END_Comment@@@

@BEG_Body
@TL(6)
IF NOT mbInit THEN RETURN; END_IF;

miActElement := miLowBound;
Element := mListStruct.List[miLowBound];

@END_Body

@@@BEG_Comment@@@
@TL(0)

@@@END_Comment@@@

@BEG_Body
@TL(9)
IF NOT mbInit THEN RETURN; END_IF;

IF miActElement < miHighBound THEN

    miActElement := miActElement + 1;
    iPos := miActElement;
    Element := mListStruct.List[miActElement];
END_IF;

@END_Body

@@@BEG_Comment@@@
@TL(0)

@@@END_Comment@@@

@BEG_Body
@TL(6)
IF NOT mbInit THEN RETURN; END_IF;

miActElement := miNextFree - 1;
Element := mListStruct.List[miActElement];

@END_Body

@@@BEG_Comment@@@
@TL(0)

@@@END_Comment@@@

@BEG_Body
@TL(9)
IF NOT mbInit THEN RETURN; END_IF;

IF miActElement > miLowBound THEN

    miActElement := miActElement - 1;
    iPos := miActElement;
    Element := mListStruct.List[miActElement];
END_IF;

@END_Body

@@@BEG_Comment@@@
@TL(0)

@@@END_Comment@@@

@BEG_Body
@TL(16)
IF NOT mbInit THEN RETURN; END_IF;

miLastFound := miLowBound;
miActElement := miLowBound;
miNextFree := miLowBound;
mListStruct :=  ListStruct;

//cheching used elements
FOR i := miLowBound TO miHighBound DO

   IF NOT mListStruct.Used[i] THEN
        miNextFree := i;
        RETURN;
   END_IF;
END_FOR;

@END_Body

@@@BEG_Comment@@@
@TL(0)

@@@END_Comment@@@

@BEG_Body
@TL(4)
IF NOT mbInit THEN RETURN; END_IF;

ListStruct := mListStruct;

@END_Body

@@@BEG_Comment@@@
@TL(0)

@@@END_Comment@@@
@END_Body

@END_Contents

(* ---- ABEmergencyStop.pu ---- *)
(*
@h    ! WARNING !
@h    The Kemro K2 system (including software) only meets category B according to EN 954-1,
@h    thus it is not intended for usage in safety-relevant control applications in the field
@h    of personal safety (e.g. emergency stop).
@h    To implement potentially necessary safety-relevant control tasks, always use additional
@h    external safety devices that are intended for the particular purpose, and meet the necessary
@h    functional safety.
@h    For further information see EN 954-1 (EN ISO 13849-1) and/or the K2-x00 user manual, chapter
@h    "CE conformity, directives and standards".

This block handles the emergency stop inputs.
If any emergency stop button is pressed the common emergency-stop signal sv_bEmergencyStop is set.
An according alarm is displayed if one the four supported emergency stop DI´s changes to FALSE.
This alarm leads to a stop and a lock of the motor.
Additionally all movements of all devices are locked.

*)

IMPORT_OVER_LISTFILE
 SET_ALARM
, SET_EVENT
, RESET_ALARM
, ASSERT
, cCompAll
, cAllDevIndex
, cMoveAll
, nLockAbort
, nUnlock
, tsTraceLevel
, tevEmergencyStop
, tevEmergencyStopData
, tnLockUnlock
, FBLockUnlock
, FBDebugTrace

END_IMPORT

ALGORITHM_BLOCK ABEmergencyStop #DUMMY_EDIT_BLOCK

SYSTEM_VAR
 sv_TraceLevel : tsTraceLevel;
 sv_bInitDone : BOOL;
 di_EmergencyStop1 : BOOL;
 di_EmergencyStop2 : BOOL;
 di_EmergencyStop3 : BOOL;
 di_EmergencyStop4 : BOOL;
 sv_bEmergencyStop : BOOL;
END_VAR

SYSTEM_OBJECT
 PU_Task_3 : TASK;
 EV_Task_3 : TASK;
 evEmergencyStop : tevEmergencyStop;
 erEmergencyStop : ALARM;
 erAssert : ALARM;
END_OBJECT

VAR
 mbLock : BOOL;
END_VAR

(*
Helper for pInputChanged.
*)

ALGORITHM aCheckInput

VAR_INPUT
 bInput : BOOL (* HW input *);
 iId : DINT (* number of emergency stop *);
END_VAR

VAR_IN_OUT
 bEventSent : BOOL;
END_VAR

VAR_TEMP
 evEmergencyStopData : tevEmergencyStopData;
END_VAR
#BEGIN_EDIT_BLOCK
(**************************************** WARNING ********************************************
 *** The KEBA Kemro K2 System including software is not intended for safety control tasks! ***
 ***                       For further information see Comment tab!                        ***
 *********************************************************************************************)

IF NOT bInput AND NOT bEventSent THEN
   //lock all movements
   SET_ALARM(Name := erEmergencyStop, SubID1 := iId);

   //fire emergencystop-event
   evEmergencyStopData.bActive := TRUE;
   SET_EVENT(evEmergencyStop, evEmergencyStopData);
   bEventSent := TRUE;
   mbLock := TRUE;
ELSIF bInput AND bEventSent THEN
   //unlock all movements
   RESET_ALARM(Name := erEmergencyStop, SubID1 := iId);

   //fire emergencystop-event
   evEmergencyStopData.bActive := FALSE;
   SET_EVENT(evEmergencyStop, evEmergencyStopData);
   bEventSent := FALSE;
END_IF;

;#END_EDIT_BLOCK END_ALGORITHM

POSTUPDATE_ALGORITHM pInputChanged ON PU_Task_3 WITH sv_bInitDone,di_EmergencyStop1,di_EmergencyStop2,di_EmergencyStop3,di_EmergencyStop4

VAR
 bFirstRunDone : BOOL (* flag to avoid unnecessary unlock events after startup *);
 bIsLinked1 : BOOL;
 bIsLinked2 : BOOL;
 bIsLinked3 : BOOL;
 bIsLinked4 : BOOL;
 bEventSent1 : BOOL;
 bEventSent2 : BOOL;
 bEventSent3 : BOOL;
 bEventSent4 : BOOL;
 nMode : tnLockUnlock;
 fbLockUnlock : FBLockUnlock;
END_VAR
#BEGIN_EDIT_BLOCK
(**************************************** WARNING ********************************************
 *** The KEBA Kemro K2 System including software is not intended for safety control tasks! ***
 ***                       For further information see Comment tab!                        ***
 *********************************************************************************************)

IF (NOT bFirstRunDone) THEN
   bIsLinked1 := IS_LINKED(di_EmergencyStop1);
   bIsLinked2 := IS_LINKED(di_EmergencyStop2);
   bIsLinked3 := IS_LINKED(di_EmergencyStop3);
   bIsLinked4 := IS_LINKED(di_EmergencyStop4);

   fbLockUnlock.DeviceId.CompId  := cCompAll;
   fbLockUnlock.DeviceId.IndexId := cAllDevIndex;
   fbLockUnlock.MoveDir := cMoveAll;
   fbLockUnlock.MoveId  := cMoveAll;
END_IF;

IF sv_bInitDone THEN
   mbLock := FALSE;

   IF bIsLinked1 THEN
      aCheckInput(bInput := di_EmergencyStop1, iId := 1, bEventSent := bEventSent1);
   END_IF;
   IF bIsLinked2 THEN
      aCheckInput(bInput := di_EmergencyStop2, iId := 2, bEventSent := bEventSent2);
   END_IF;
   IF bIsLinked3 THEN
      aCheckInput(bInput := di_EmergencyStop3, iId := 3, bEventSent := bEventSent3);
   END_IF;
   IF bIsLinked4 THEN
      aCheckInput(bInput := di_EmergencyStop4, iId := 4, bEventSent := bEventSent4);
   END_IF;

   IF mbLock THEN
      nMode := nLockAbort;
   ELSE
      nMode := nUnlock;
   END_IF;

   //lock/unlock all movements
   IF (nMode = nLockAbort OR bFirstRunDone) THEN
      fbLockUnlock(Mode := nMode);
   END_IF;

   bFirstRunDone := TRUE;
END_IF;

;#END_EDIT_BLOCK END_ALGORITHM

(*
This eventalgo receives the emergency-stop event.
If any emergencystop button is pressed the common emergency-stop signal sv_bEmergencyStop is set.
The event must be sent from each emergency-stop handler. eg. OperationMode, Robot interface
*)

EVENT_ALGORITHM evaEmergencyStop ON EV_Task_3 WITH evEmergencyStop

VAR_INPUT
 evEmergencyStopData : tevEmergencyStopData;
END_VAR

VAR
 iEmgStopActive : DINT;
 fbDebugTrace : FBDebugTrace;
 bTmp : BOOL;
END_VAR
#BEGIN_EDIT_BLOCK
(**************************************** WARNING ********************************************
 *** The KEBA Kemro K2 System including software is not intended for safety control tasks! ***
 ***                       For further information see Comment tab!                        ***
 *********************************************************************************************)

IF evEmergencyStopData.bActive THEN
   iEmgStopActive := iEmgStopActive + 1;
ELSIF iEmgStopActive > 0 THEN
   iEmgStopActive := iEmgStopActive - 1;
ELSIF sv_TraceLevel.bApplication THEN
   // an event with status bActive=FALSE was received eventhough no emergency stop was active
   fbDebugTrace(sText := 'ABEmergencyStop.evaEmergencyStop: error: invalid event received');
   bTmp := ASSERT(FALSE, erAssert);
END_IF;
// if any emergency stop is pressed the common signal is set
sv_bEmergencyStop := iEmgStopActive > 0;

;#END_EDIT_BLOCK END_ALGORITHM

END_ALGORITHM_BLOCK

#END_OF_IEC_PART

@Puma @IecEditor 6 114 @Pou 25
@@@BEG_Comment@@@
@h    ! WARNING !
@h    The Kemro K2 system (including software) only meets category B according to EN 954-1,
@h    thus it is not intended for usage in safety-relevant control applications in the field
@h    of personal safety (e.g. emergency stop).
@h    To implement potentially necessary safety-relevant control tasks, always use additional
@h    external safety devices that are intended for the particular purpose, and meet the necessary
@h    functional safety.
@h    For further information see EN 954-1 (EN ISO 13849-1) and/or the K2-x00 user manual, chapter
@h    "CE conformity, directives and standards".

This block handles the emergency stop inputs.
If any emergency stop button is pressed the common emergency-stop signal sv_bEmergencyStop is set.
An according alarm is displayed if one the four supported emergency stop DI´s changes to FALSE.
This alarm leads to a stop and a lock of the motor.
Additionally all movements of all devices are locked.

@@@END_Comment@@@

@BEG_Contents

@BEG_Func
@RT(17)FuncTreeContainer
4
@Var @RT(9)SET_ALARM @RT(0) @T @T @DERIVED 0 @F @RT(23)KEBA_STANDARD_PROCEDURE @F
@T
@BEG_Attrib
0 @RT(0) @RT(0)
@END_Attrib
1 1 @F @F @F @F

@Var @RT(9)SET_EVENT @RT(0) @T @T @DERIVED 0 @F @RT(23)KEBA_STANDARD_PROCEDURE @F
@T
@BEG_Attrib
0 @RT(0) @RT(0)
@END_Attrib
1 1 @F @F @F @F

@Var @RT(11)RESET_ALARM @RT(0) @T @T @DERIVED 0 @F @RT(23)KEBA_STANDARD_PROCEDURE @F
@T
@BEG_Attrib
0 @RT(0) @RT(0)
@END_Attrib
1 1 @F @F @F @F

@Var @RT(6)ASSERT @RT(0) @T @T @DERIVED 0 @F @RT(8)FUNCTION @F
@T
@BEG_Attrib
0 @RT(0) @RT(0)
@END_Attrib
1 1 @F @F @F @F

@END_Func

@BEG_Const
@RT(18)ConstTreeContainer
5
@Var @RT(8)cCompAll @RT(0) @T @F @DT @RT(4)DINT @RT(0) @T @T @BASIC 0 @F
@F @F
@T
@BEG_Attrib
0 @RT(10)cMaxCompId @RT(22)to lock all components
@END_Attrib
1 1 @F @F @F @F

@Var @RT(12)cAllDevIndex @RT(0) @T @F @DT @RT(4)DINT @RT(0) @T @T @BASIC 0 @F
@F @F
@T
@BEG_Attrib
0 @RT(2)11 @RT(59)to lock all devices of a component ( = cMaxDeviceIndex + 1)
@END_Attrib
1 1 @F @F @F @F

@Var @RT(8)cMoveAll @RT(0) @T @F @DT @RT(4)DINT @RT(0) @T @T @BASIC 0 @F
@F @F
@T
@BEG_Attrib
0 @RT(13)cMaxMoveIdent @RT(32)all movements (for evLockUnlock)
@END_Attrib
1 1 @F @F @F @F

@Var @RT(10)nLockAbort @RT(0) @T @T @DERIVED 0 @F @RT(12)tnLockUnlock @F
@T
@BEG_Attrib
0 @RT(1)0 @RT(0)
@END_Attrib
1 1 @F @F @F @F

@Var @RT(7)nUnlock @RT(0) @T @T @DERIVED 0 @F @RT(12)tnLockUnlock @F
@T
@BEG_Attrib
0 @RT(1)2 @RT(0)
@END_Attrib
1 1 @F @F @F @F

@END_Const

@BEG_Export

@BEG_Kind
@ALGORITHM_BLOCK @RT(15)ABEmergencyStop @STRUCTURED_TEXT
@RT(0) @RT(0) @RT(0)
@END_Kind

@BEG_Dcl
@RT(16)DclTreeContainer
13
@Var @RT(13)sv_TraceLevel @RT(0) @T @T @DERIVED 0 @T @T @DT @RT(12)tsTraceLevel @RT(0) @T @T @UNKNOWN 0 @F
@F @F
@T
@BEG_Attrib
3 @RT(0) @RT(0) @RT(0)
@END_Attrib
1 8 @F @F @F @F

@Var @RT(12)sv_bInitDone @RT(0) @T @F @DT @RT(4)BOOL @RT(0) @T @T @BASIC 0 @F
@F @F
@T
@BEG_Attrib
3 @RT(0) @RT(0) @RT(0)
@END_Attrib
1 8 @F @F @F @F

@Var @RT(17)di_EmergencyStop1 @RT(0) @T @F @DT @RT(4)BOOL @RT(0) @T @T @BASIC 0 @F
@F @F
@T
@BEG_Attrib
3 @RT(0) @RT(0) @RT(0)
@END_Attrib
1 8 @F @F @F @F

@Var @RT(17)di_EmergencyStop2 @RT(0) @T @F @DT @RT(4)BOOL @RT(0) @T @T @BASIC 0 @F
@F @F
@T
@BEG_Attrib
3 @RT(0) @RT(0) @RT(0)
@END_Attrib
1 8 @F @F @F @F

@Var @RT(17)di_EmergencyStop3 @RT(0) @T @F @DT @RT(4)BOOL @RT(0) @T @T @BASIC 0 @F
@F @F
@T
@BEG_Attrib
3 @RT(0) @RT(0) @RT(0)
@END_Attrib
1 8 @F @F @F @F

@Var @RT(17)di_EmergencyStop4 @RT(0) @T @F @DT @RT(4)BOOL @RT(0) @T @T @BASIC 0 @F
@F @F
@T
@BEG_Attrib
3 @RT(0) @RT(0) @RT(0)
@END_Attrib
1 8 @F @F @F @F

@Var @RT(17)sv_bEmergencyStop @RT(0) @T @F @DT @RT(4)BOOL @RT(0) @T @T @BASIC 0 @F
@F @F
@T
@BEG_Attrib
3 @RT(0) @RT(0) @RT(0)
@END_Attrib
1 8 @F @F @F @F

@Var @RT(9)PU_Task_3 @RT(0) @T @F @DT @RT(4)TASK @RT(0) @T @T @BASIC 0 @F
@F @F
@T
@BEG_Attrib
3 @RT(0) @RT(0) @RT(0)
@END_Attrib
1 7 @F @F @F @F

@Var @RT(9)EV_Task_3 @RT(0) @T @F @DT @RT(4)TASK @RT(0) @T @T @BASIC 0 @F
@F @F
@T
@BEG_Attrib
3 @RT(0) @RT(0) @RT(0)
@END_Attrib
1 7 @F @F @F @F

@Var @RT(15)evEmergencyStop @RT(0) @T @T @DERIVED 0 @T @T @DT @RT(16)tevEmergencyStop @RT(0) @T @T @UNKNOWN 0 @F
@F @F
@T
@BEG_Attrib
3 @RT(0) @RT(0) @RT(0)
@END_Attrib
1 7 @F @F @F @F

@Var @RT(15)erEmergencyStop @RT(0) @T @F @DT @RT(5)ALARM @RT(0) @T @T @BASIC 0 @F
@F @F
@T
@BEG_Attrib
3 @RT(0) @RT(0) @RT(0)
@END_Attrib
1 7 @F @F @F @F

@Var @RT(8)erAssert @RT(0) @T @F @DT @RT(5)ALARM @RT(0) @T @T @BASIC 0 @F
@F @F
@T
@BEG_Attrib
3 @RT(0) @RT(0) @RT(0)
@END_Attrib
1 7 @F @F @F @F

@Var @RT(6)mbLock @RT(0) @T @F @DT @RT(4)BOOL @RT(0) @T @T @BASIC 0 @F
@F @F
@T
@BEG_Attrib
3 @RT(0) @RT(0) @RT(0)
@END_Attrib
1 0 @F @F @F @F

@END_Dcl

@END_Export

@BEG_Body

3

@BEG_Export

@BEG_Algo
@ALGORITHM @RT(11)aCheckInput @STRUCTURED_TEXT
@RT(0) @RT(0) @RT(0) @F @F
@END_Algo

@BEG_Dcl
@RT(16)DclTreeContainer
4
@Var @RT(6)bInput @RT(0) @T @F @DT @RT(4)BOOL @RT(0) @T @T @BASIC 0 @F
@F @F
@T
@BEG_Attrib
3 @RT(0) @RT(8)HW input @RT(0)
@END_Attrib
1 1 @F @F @F @F

@Var @RT(3)iId @RT(0) @T @F @DT @RT(4)DINT @RT(0) @T @T @BASIC 0 @F
@F @F
@T
@BEG_Attrib
3 @RT(0) @RT(24)number of emergency stop @RT(0)
@END_Attrib
1 1 @F @F @F @F

@Var @RT(10)bEventSent @RT(0) @T @F @DT @RT(4)BOOL @RT(0) @T @T @BASIC 0 @F
@F @F
@T
@BEG_Attrib
3 @RT(0) @RT(0) @RT(0)
@END_Attrib
1 2 @F @F @F @F

@Var @RT(19)evEmergencyStopData @RT(0) @T @T @DERIVED 0 @F @RT(20)tevEmergencyStopData @F
@T
@BEG_Attrib
3 @RT(0) @RT(0) @RT(0)
@END_Attrib
1 4 @F @F @F @F

@END_Dcl

@END_Export

@BEG_Export

@BEG_Algo
@POSTUPDATE_ALGORITHM @RT(13)pInputChanged @STRUCTURED_TEXT
@RT(0) @RT(84)sv_bInitDone,di_EmergencyStop1,di_EmergencyStop2,di_EmergencyStop3,di_EmergencyStop4 @RT(9)PU_Task_3 @F @F
@END_Algo

@BEG_Dcl
@RT(16)DclTreeContainer
11
@Var @RT(13)bFirstRunDone @RT(0) @T @F @DT @RT(4)BOOL @RT(0) @T @T @BASIC 0 @F
@F @F
@T
@BEG_Attrib
3 @RT(0) @RT(53)flag to avoid unnecessary unlock events after startup @RT(0)
@END_Attrib
1 0 @F @F @F @F

@Var @RT(10)bIsLinked1 @RT(0) @T @F @DT @RT(4)BOOL @RT(0) @T @T @BASIC 0 @F
@F @F
@T
@BEG_Attrib
3 @RT(0) @RT(0) @RT(0)
@END_Attrib
1 0 @F @F @F @F

@Var @RT(10)bIsLinked2 @RT(0) @T @F @DT @RT(4)BOOL @RT(0) @T @T @BASIC 0 @F
@F @F
@T
@BEG_Attrib
3 @RT(0) @RT(0) @RT(0)
@END_Attrib
1 0 @F @F @F @F

@Var @RT(10)bIsLinked3 @RT(0) @T @F @DT @RT(4)BOOL @RT(0) @T @T @BASIC 0 @F
@F @F
@T
@BEG_Attrib
3 @RT(0) @RT(0) @RT(0)
@END_Attrib
1 0 @F @F @F @F

@Var @RT(10)bIsLinked4 @RT(0) @T @F @DT @RT(4)BOOL @RT(0) @T @T @BASIC 0 @F
@F @F
@T
@BEG_Attrib
3 @RT(0) @RT(0) @RT(0)
@END_Attrib
1 0 @F @F @F @F

@Var @RT(11)bEventSent1 @RT(0) @T @F @DT @RT(4)BOOL @RT(0) @T @T @BASIC 0 @F
@F @F
@T
@BEG_Attrib
3 @RT(0) @RT(0) @RT(0)
@END_Attrib
1 0 @F @F @F @F

@Var @RT(11)bEventSent2 @RT(0) @T @F @DT @RT(4)BOOL @RT(0) @T @T @BASIC 0 @F
@F @F
@T
@BEG_Attrib
3 @RT(0) @RT(0) @RT(0)
@END_Attrib
1 0 @F @F @F @F

@Var @RT(11)bEventSent3 @RT(0) @T @F @DT @RT(4)BOOL @RT(0) @T @T @BASIC 0 @F
@F @F
@T
@BEG_Attrib
3 @RT(0) @RT(0) @RT(0)
@END_Attrib
1 0 @F @F @F @F

@Var @RT(11)bEventSent4 @RT(0) @T @F @DT @RT(4)BOOL @RT(0) @T @T @BASIC 0 @F
@F @F
@T
@BEG_Attrib
3 @RT(0) @RT(0) @RT(0)
@END_Attrib
1 0 @F @F @F @F

@Var @RT(5)nMode @RT(0) @T @T @DERIVED 0 @T @T @DT @RT(12)tnLockUnlock @RT(0) @T @T @UNKNOWN 0 @F
@F @F
@T
@BEG_Attrib
3 @RT(0) @RT(0) @RT(0)
@END_Attrib
1 0 @F @F @F @F

@Var @RT(12)fbLockUnlock @RT(0) @T @T @DERIVED 0 @T @T @DT @RT(12)FBLockUnlock @RT(0) @T @T @UNKNOWN 0 @F
@F @F
@T
@BEG_Attrib
3 @RT(0) @RT(0) @RT(0)
@END_Attrib
1 0 @F @F @F @F

@END_Dcl

@END_Export

@BEG_Export

@BEG_Algo
@EVENT_ALGORITHM @RT(16)evaEmergencyStop @STRUCTURED_TEXT
@RT(0) @RT(15)evEmergencyStop @RT(9)EV_Task_3 @F @F
@END_Algo

@BEG_Dcl
@RT(16)DclTreeContainer
4
@Var @RT(19)evEmergencyStopData @RT(0) @T @T @DERIVED 0 @F @RT(20)tevEmergencyStopData @F
@T
@BEG_Attrib
3 @RT(0) @RT(0) @RT(0)
@END_Attrib
1 1 @F @F @F @F

@Var @RT(14)iEmgStopActive @RT(0) @T @F @DT @RT(4)DINT @RT(0) @T @T @BASIC 0 @F
@F @F
@T
@BEG_Attrib
3 @RT(0) @RT(0) @RT(0)
@END_Attrib
1 0 @F @F @F @F

@Var @RT(12)fbDebugTrace @RT(0) @T @T @DERIVED 0 @T @T @DT @RT(12)FBDebugTrace @RT(0) @T @T @UNKNOWN 0 @F
@F @F
@T
@BEG_Attrib
3 @RT(0) @RT(0) @RT(0)
@END_Attrib
1 0 @F @F @F @F

@Var @RT(4)bTmp @RT(0) @T @F @DT @RT(4)BOOL @RT(0) @T @T @BASIC 0 @F
@F @F
@T
@BEG_Attrib
3 @RT(0) @RT(0) @RT(0)
@END_Attrib
1 0 @F @F @F @F

@END_Dcl

@END_Export

@BEG_Body
@TL(24)
(**************************************** WARNING ********************************************
 *** The KEBA Kemro K2 System including software is not intended for safety control tasks! ***
 ***                       For further information see Comment tab!                        ***
 *********************************************************************************************)

IF NOT bInput AND NOT bEventSent THEN
   //lock all movements
   SET_ALARM(Name := erEmergencyStop, SubID1 := iId);

   //fire emergencystop-event
   evEmergencyStopData.bActive := TRUE;
   SET_EVENT(evEmergencyStop, evEmergencyStopData);
   bEventSent := TRUE;
   mbLock := TRUE;
ELSIF bInput AND bEventSent THEN
   //unlock all movements
   RESET_ALARM(Name := erEmergencyStop, SubID1 := iId);

   //fire emergencystop-event
   evEmergencyStopData.bActive := FALSE;
   SET_EVENT(evEmergencyStop, evEmergencyStopData);
   bEventSent := FALSE;
END_IF;

@END_Body

@@@BEG_Comment@@@
@TL(1)
Helper for pInputChanged.
@@@END_Comment@@@

@BEG_Body
@TL(48)
(**************************************** WARNING ********************************************
 *** The KEBA Kemro K2 System including software is not intended for safety control tasks! ***
 ***                       For further information see Comment tab!                        ***
 *********************************************************************************************)

IF (NOT bFirstRunDone) THEN
   bIsLinked1 := IS_LINKED(di_EmergencyStop1);
   bIsLinked2 := IS_LINKED(di_EmergencyStop2);
   bIsLinked3 := IS_LINKED(di_EmergencyStop3);
   bIsLinked4 := IS_LINKED(di_EmergencyStop4);

   fbLockUnlock.DeviceId.CompId  := cCompAll;
   fbLockUnlock.DeviceId.IndexId := cAllDevIndex;
   fbLockUnlock.MoveDir := cMoveAll;
   fbLockUnlock.MoveId  := cMoveAll;
END_IF;

IF sv_bInitDone THEN
   mbLock := FALSE;

   IF bIsLinked1 THEN
      aCheckInput(bInput := di_EmergencyStop1, iId := 1, bEventSent := bEventSent1);
   END_IF;
   IF bIsLinked2 THEN
      aCheckInput(bInput := di_EmergencyStop2, iId := 2, bEventSent := bEventSent2);
   END_IF;
   IF bIsLinked3 THEN
      aCheckInput(bInput := di_EmergencyStop3, iId := 3, bEventSent := bEventSent3);
   END_IF;
   IF bIsLinked4 THEN
      aCheckInput(bInput := di_EmergencyStop4, iId := 4, bEventSent := bEventSent4);
   END_IF;

   IF mbLock THEN
      nMode := nLockAbort;
   ELSE
      nMode := nUnlock;
   END_IF;

   //lock/unlock all movements
   IF (nMode = nLockAbort OR bFirstRunDone) THEN
      fbLockUnlock(Mode := nMode);
   END_IF;

   bFirstRunDone := TRUE;
END_IF;

@END_Body

@@@BEG_Comment@@@
@TL(0)

@@@END_Comment@@@

@BEG_Body
@TL(17)
(**************************************** WARNING ********************************************
 *** The KEBA Kemro K2 System including software is not intended for safety control tasks! ***
 ***                       For further information see Comment tab!                        ***
 *********************************************************************************************)

IF evEmergencyStopData.bActive THEN
   iEmgStopActive := iEmgStopActive + 1;
ELSIF iEmgStopActive > 0 THEN
   iEmgStopActive := iEmgStopActive - 1;
ELSIF sv_TraceLevel.bApplication THEN
   // an event with status bActive=FALSE was received eventhough no emergency stop was active
   fbDebugTrace(sText := 'ABEmergencyStop.evaEmergencyStop: error: invalid event received');
   bTmp := ASSERT(FALSE, erAssert);
END_IF;
// if any emergency stop is pressed the common signal is set
sv_bEmergencyStop := iEmgStopActive > 0;

@END_Body

@@@BEG_Comment@@@
@TL(3)
This eventalgo receives the emergency-stop event.
If any emergencystop button is pressed the common emergency-stop signal sv_bEmergencyStop is set.
The event must be sent from each emergency-stop handler. eg. OperationMode, Robot interface
@@@END_Comment@@@
@END_Body

@END_Contents

(* ---- ABEventNotification.pu ---- *)
IMPORT_OVER_LISTFILE
 SET_EVENT
, STATE_ALARM
, tevRequestEventNotification
, RTC
, tevUpdateEventNotification
, tevEventNotificationData
, tevAlarmConfirm
, tnOperationMode
, ALARM_STATE_DATA
, tevAlarmConfirmData

END_IMPORT

ALGORITHM_BLOCK ABEventNotification #DUMMY_EDIT_BLOCK

SYSTEM_VAR
 sv_rProdTimeRemaining : REAL;
 sv_bUseProdCounter : BOOL (* use shot counter *);
 sv_iProdCounterRemaining : DINT;
 sv_iProdCounterAct : DINT;
 sv_OperationMode : tnOperationMode;
END_VAR

SYSTEM_OBJECT
 PU_Task_13 : TASK;
 evRequestEventNotification : tevRequestEventNotification;
 evUpdateEventNotification : tevUpdateEventNotification;
 erProdLimitReached : ALARM;
 evAlarmConfirm : tevAlarmConfirm;
END_OBJECT

VAR
 fbRTC : RTC;
 eventNotificationData : tevEventNotificationData := (iType:=cEvNotificationType_Production,iInstance:=1);
 mbProdEvNotificationActive : BOOL;
END_VAR

ALGORITHM aCheckAndSendUpdate

VAR
 dEstimatedExpirationDate : DATE_AND_TIME := cUTCZeroDate;
 dLastEstimatedExpirationDate : DATE_AND_TIME := cUTCZeroDate;
 dTimeDifference : TIME;
END_VAR

VAR CONSTANT
 dEstimationTolerance : TIME := T#30s;
END_VAR
#BEGIN_EDIT_BLOCK
(**************************************** WARNING ********************************************
 *** The KEBA Kemro K2 System including software is not intended for safety control tasks! ***
 ***                       For further information see Comment tab!                        ***
 *********************************************************************************************)

// Estimate expiration date and send event notification update if necessary
fbRTC();

// Calculate estimated expiration date depending on remaining production time
dEstimatedExpirationDate := fbRTC.CDT + T#1h * sv_rProdTimeRemaining;

// Calculate a positive time difference
dTimeDifference := dEstimatedExpirationDate - dLastEstimatedExpirationDate;
IF dTimeDifference < T#0s THEN
    dTimeDifference := dTimeDifference * -1;
END_IF;

IF sv_bUseProdCounter
    AND (sv_OperationMode >= nHalfAutomatic)
    AND NOT (sv_iProdCounterAct = 0 AND sv_iProdCounterRemaining = 0)
    AND ((dTimeDifference >= dEstimationTolerance) OR NOT mbProdEvNotificationActive) THEN

    // Valid production settings and new estimated expiration date differs from last calculated expiration date
    // -> Send event notification update
    eventNotificationData.dExpirationDate := dEstimatedExpirationDate;

    mbProdEvNotificationActive := TRUE;

    // Send event notification update
    SET_EVENT(evUpdateEventNotification, eventNotificationData);
END_IF;

dLastEstimatedExpirationDate := dEstimatedExpirationDate;

;#END_EDIT_BLOCK END_ALGORITHM

EVENT_ALGORITHM evaRequestEventNotification ON PU_Task_13 WITH evRequestEventNotification

#BEGIN_EDIT_BLOCK
(**************************************** WARNING ********************************************
 *** The KEBA Kemro K2 System including software is not intended for safety control tasks! ***
 ***                       For further information see Comment tab!                        ***
 *********************************************************************************************)

// Reset active flag
mbProdEvNotificationActive := FALSE;

// Send update for all production event notifications
aCheckAndSendUpdate();

;#END_EDIT_BLOCK END_ALGORITHM

POSTUPDATE_ALGORITHM pProdSettingsChanged ON PU_Task_13 WITH sv_OperationMode, sv_iProdCounterRemaining, sv_bUseProdCounter

VAR
 State : ALARM_STATE_DATA;
END_VAR
#BEGIN_EDIT_BLOCK
(**************************************** WARNING ********************************************
 *** The KEBA Kemro K2 System including software is not intended for safety control tasks! ***
 ***                       For further information see Comment tab!                        ***
 *********************************************************************************************)

IF mbProdEvNotificationActive
    AND (NOT sv_bUseProdCounter
         OR (sv_iProdCounterAct = 0 AND sv_iProdCounterRemaining = 0)
         OR (sv_OperationMode < nHalfAutomatic)) THEN

    // Check state of "production limit reached"-alarm
    STATE_ALARM(Name := erProdLimitReached,
            State := State);

    IF State.ALARM_STATE = ALARM_STATE_INACTIVE_ACK THEN
        // Production counter is not used any more
        // or shot counter was reset
        // or production has stopped and alarm is not active any more
        // -> Invalidate event notification
        mbProdEvNotificationActive := FALSE;

        eventNotificationData.dExpirationDate := cUTCZeroDate;
        SET_EVENT(evUpdateEventNotification, eventNotificationData);
        RETURN;
    END_IF;
END_IF;

aCheckAndSendUpdate();

;#END_EDIT_BLOCK END_ALGORITHM

EVENT_ALGORITHM evaAlarmConfirm ON PU_Task_13 WITH evAlarmConfirm

VAR_INPUT
 evAlarmConfirmData : tevAlarmConfirmData;
END_VAR

VAR
 State : ALARM_STATE_DATA;
END_VAR
#BEGIN_EDIT_BLOCK
(**************************************** WARNING ********************************************
 *** The KEBA Kemro K2 System including software is not intended for safety control tasks! ***
 ***                       For further information see Comment tab!                        ***
 *********************************************************************************************)

IF mbProdEvNotificationActive AND sv_iProdCounterRemaining = 0 THEN
    // Check state of "production limit reached"-alarm
    STATE_ALARM(Name := erProdLimitReached,
            State := State);

    IF State.ALARM_STATE = ALARM_STATE_INACTIVE_ACK THEN
        // Alarm inactive and quitted
        // -> Invalidate event notification
        mbProdEvNotificationActive := FALSE;
        eventNotificationData.dExpirationDate := cUTCZeroDate;
        SET_EVENT(evUpdateEventNotification, eventNotificationData);
    END_IF;
END_IF;

;#END_EDIT_BLOCK END_ALGORITHM

END_ALGORITHM_BLOCK

#END_OF_IEC_PART

@Puma @IecEditor 6 131 @Pou 25
@@@BEG_Comment@@@

@@@END_Comment@@@

@BEG_Contents

@BEG_Func
@RT(17)FuncTreeContainer
2
@Var @RT(9)SET_EVENT @RT(0) @T @T @DERIVED 0 @F @RT(23)KEBA_STANDARD_PROCEDURE @F
@T
@BEG_Attrib
0 @RT(0) @RT(0)
@END_Attrib
1 1 @F @F @F @F

@Var @RT(11)STATE_ALARM @RT(0) @T @T @DERIVED 0 @F @RT(23)KEBA_STANDARD_PROCEDURE @F
@T
@BEG_Attrib
0 @RT(0) @RT(0)
@END_Attrib
1 1 @F @F @F @F

@END_Func

@BEG_Const
@RT(18)ConstTreeContainer
0
@END_Const

@BEG_Export

@BEG_Kind
@ALGORITHM_BLOCK @RT(19)ABEventNotification @STRUCTURED_TEXT
@RT(0) @RT(0) @RT(0)
@END_Kind

@BEG_Dcl
@RT(16)DclTreeContainer
13
@Var @RT(10)PU_Task_13 @RT(0) @T @T @RENAMED 0 @T @T @DT @RT(4)TASK @RT(0) @T @T @BASIC 0 @F
@F @F
@T
@BEG_Attrib
3 @RT(0) @RT(0) @RT(0)
@END_Attrib
1 7 @F @F @F @F

@Var @RT(26)evRequestEventNotification @RT(0) @T @T @DERIVED 0 @T @T @DT @RT(27)tevRequestEventNotification @RT(0) @T @T @UNKNOWN 0 @F
@F @F
@T
@BEG_Attrib
3 @RT(0) @RT(0) @RT(0)
@END_Attrib
1 7 @F @F @F @F

@Var @RT(5)fbRTC @RT(0) @T @T @DERIVED 0 @T @T @DT @RT(3)RTC @RT(0) @T @T @UNKNOWN 0 @F
@F @F
@T
@BEG_Attrib
3 @RT(0) @RT(0) @RT(0)
@END_Attrib
1 0 @F @F @F @F

@Var @RT(25)evUpdateEventNotification @RT(0) @T @T @DERIVED 0 @T @T @DT @RT(26)tevUpdateEventNotification @RT(0) @T @T @UNKNOWN 0 @F
@F @F
@T
@BEG_Attrib
3 @RT(0) @RT(0) @RT(0)
@END_Attrib
1 7 @F @F @F @F

@Var @RT(21)sv_rProdTimeRemaining @RT(0) @T @F @DT @RT(4)REAL @RT(0) @T @T @BASIC 0 @F
@F @F
@T
@BEG_Attrib
3 @RT(0) @RT(0) @RT(0)
@END_Attrib
1 8 @F @F @F @F

@Var @RT(18)sv_bUseProdCounter @RT(0) @T @F @DT @RT(4)BOOL @RT(0) @T @T @BASIC 0 @F
@F @F
@T
@BEG_Attrib
3 @RT(0) @RT(16)use shot counter @RT(0)
@END_Attrib
1 8 @F @F @F @F

@Var @RT(21)eventNotificationData @RT(0) @T @T @DERIVED 0 @T @T @DT @RT(24)tevEventNotificationData @RT(0) @T @T @UNKNOWN 0 @F
@F @F
@T
@BEG_Attrib
3 @RT(52)(iType:=cEvNotificationType_Production,iInstance:=1) @RT(0) @RT(0)
@END_Attrib
1 0 @F @F @F @F

@Var @RT(18)erProdLimitReached @RT(0) @T @F @DT @RT(5)ALARM @RT(0) @T @T @BASIC 0 @F
@F @F
@T
@BEG_Attrib
3 @RT(0) @RT(0) @RT(0)
@END_Attrib
1 7 @F @F @F @F

@Var @RT(14)evAlarmConfirm @RT(0) @T @T @DERIVED 0 @T @T @DT @RT(15)tevAlarmConfirm @RT(0) @T @T @UNKNOWN 0 @F
@F @F
@T
@BEG_Attrib
3 @RT(0) @RT(0) @RT(0)
@END_Attrib
1 7 @F @F @F @F

@Var @RT(24)sv_iProdCounterRemaining @RT(0) @T @F @DT @RT(4)DINT @RT(0) @T @T @BASIC 0 @F
@F @F
@T
@BEG_Attrib
3 @RT(0) @RT(0) @RT(0)
@END_Attrib
1 8 @F @F @F @F

@Var @RT(18)sv_iProdCounterAct @RT(0) @T @F @DT @RT(4)DINT @RT(0) @T @T @BASIC 0 @F
@F @F
@T
@BEG_Attrib
3 @RT(0) @RT(0) @RT(0)
@END_Attrib
1 8 @F @F @F @F

@Var @RT(16)sv_OperationMode @RT(0) @T @T @DERIVED 0 @T @T @DT @RT(15)tnOperationMode @RT(0) @T @T @UNKNOWN 0 @F
@F @F
@T
@BEG_Attrib
3 @RT(0) @RT(0) @RT(0)
@END_Attrib
1 8 @F @F @F @F

@Var @RT(26)mbProdEvNotificationActive @RT(0) @T @F @DT @RT(4)BOOL @RT(0) @T @T @BASIC 0 @F
@F @F
@T
@BEG_Attrib
3 @RT(0) @RT(0) @RT(0)
@END_Attrib
1 0 @F @F @F @F

@END_Dcl

@END_Export

@BEG_Body

4

@BEG_Export

@BEG_Algo
@ALGORITHM @RT(19)aCheckAndSendUpdate @STRUCTURED_TEXT
@RT(0) @RT(0) @RT(0) @F @F
@END_Algo

@BEG_Dcl
@RT(16)DclTreeContainer
4
@Var @RT(24)dEstimatedExpirationDate @RT(0) @T @F @DT @RT(13)DATE_AND_TIME @RT(0) @T @T @BASIC 0 @F
@F @F
@T
@BEG_Attrib
3 @RT(12)cUTCZeroDate @RT(0) @RT(0)
@END_Attrib
1 0 @F @F @F @F

@Var @RT(28)dLastEstimatedExpirationDate @RT(0) @T @F @DT @RT(13)DATE_AND_TIME @RT(0) @T @T @BASIC 0 @F
@F @F
@T
@BEG_Attrib
3 @RT(12)cUTCZeroDate @RT(0) @RT(0)
@END_Attrib
1 0 @F @F @F @F

@Var @RT(20)dEstimationTolerance @RT(0) @T @F @DT @RT(4)TIME @RT(0) @T @T @BASIC 0 @F
@F @F
@T
@BEG_Attrib
3 @RT(5)T#30s @RT(0) @RT(0)
@END_Attrib
1 15 @F @F @F @F

@Var @RT(15)dTimeDifference @RT(0) @T @F @DT @RT(4)TIME @RT(0) @T @T @BASIC 0 @F
@F @F
@T
@BEG_Attrib
3 @RT(0) @RT(0) @RT(0)
@END_Attrib
1 0 @F @F @F @F

@END_Dcl

@END_Export

@BEG_Export

@BEG_Algo
@EVENT_ALGORITHM @RT(27)evaRequestEventNotification @STRUCTURED_TEXT
@RT(0) @RT(26)evRequestEventNotification @RT(10)PU_Task_13 @F @F
@END_Algo

@BEG_Dcl
@RT(16)DclTreeContainer
0
@END_Dcl

@END_Export

@BEG_Export

@BEG_Algo
@POSTUPDATE_ALGORITHM @RT(20)pProdSettingsChanged @STRUCTURED_TEXT
@RT(0) @RT(62)sv_OperationMode, sv_iProdCounterRemaining, sv_bUseProdCounter @RT(10)PU_Task_13 @F @F
@END_Algo

@BEG_Dcl
@RT(16)DclTreeContainer
1
@Var @RT(5)State @RT(0) @T @T @DERIVED 0 @T @T @DT @RT(16)ALARM_STATE_DATA @RT(0) @T @T @UNKNOWN 0 @F
@F @F
@T
@BEG_Attrib
3 @RT(0) @RT(0) @RT(0)
@END_Attrib
1 0 @F @F @F @F

@END_Dcl

@END_Export

@BEG_Export

@BEG_Algo
@EVENT_ALGORITHM @RT(15)evaAlarmConfirm @STRUCTURED_TEXT
@RT(0) @RT(14)evAlarmConfirm @RT(10)PU_Task_13 @F @F
@END_Algo

@BEG_Dcl
@RT(16)DclTreeContainer
2
@Var @RT(5)State @RT(0) @T @T @DERIVED 0 @T @T @DT @RT(16)ALARM_STATE_DATA @RT(0) @T @T @UNKNOWN 0 @F
@F @F
@T
@BEG_Attrib
3 @RT(0) @RT(0) @RT(0)
@END_Attrib
1 0 @F @F @F @F

@Var @RT(18)evAlarmConfirmData @RT(0) @T @T @DERIVED 0 @T @T @DT @RT(19)tevAlarmConfirmData @RT(0) @T @T @UNKNOWN 0 @F
@F @F
@T
@BEG_Attrib
3 @RT(0) @RT(0) @RT(0)
@END_Attrib
1 1 @F @F @F @F

@END_Dcl

@END_Export

@BEG_Body
@TL(34)
(**************************************** WARNING ********************************************
 *** The KEBA Kemro K2 System including software is not intended for safety control tasks! ***
 ***                       For further information see Comment tab!                        ***
 *********************************************************************************************)

// Estimate expiration date and send event notification update if necessary
fbRTC();

// Calculate estimated expiration date depending on remaining production time
dEstimatedExpirationDate := fbRTC.CDT + T#1h * sv_rProdTimeRemaining;

// Calculate a positive time difference
dTimeDifference := dEstimatedExpirationDate - dLastEstimatedExpirationDate;
IF dTimeDifference < T#0s THEN
    dTimeDifference := dTimeDifference * -1;
END_IF;

IF sv_bUseProdCounter
    AND (sv_OperationMode >= nHalfAutomatic)
    AND NOT (sv_iProdCounterAct = 0 AND sv_iProdCounterRemaining = 0)
    AND ((dTimeDifference >= dEstimationTolerance) OR NOT mbProdEvNotificationActive) THEN

    // Valid production settings and new estimated expiration date differs from last calculated expiration date
    // -> Send event notification update
    eventNotificationData.dExpirationDate := dEstimatedExpirationDate;

    mbProdEvNotificationActive := TRUE;

    // Send event notification update
    SET_EVENT(evUpdateEventNotification, eventNotificationData);
END_IF;

dLastEstimatedExpirationDate := dEstimatedExpirationDate;

@END_Body

@@@BEG_Comment@@@
@TL(0)

@@@END_Comment@@@

@BEG_Body
@TL(13)
(**************************************** WARNING ********************************************
 *** The KEBA Kemro K2 System including software is not intended for safety control tasks! ***
 ***                       For further information see Comment tab!                        ***
 *********************************************************************************************)

// Reset active flag
mbProdEvNotificationActive := FALSE;

// Send update for all production event notifications
aCheckAndSendUpdate();

@END_Body

@@@BEG_Comment@@@
@TL(0)

@@@END_Comment@@@

@BEG_Body
@TL(29)
(**************************************** WARNING ********************************************
 *** The KEBA Kemro K2 System including software is not intended for safety control tasks! ***
 ***                       For further information see Comment tab!                        ***
 *********************************************************************************************)

IF mbProdEvNotificationActive
    AND (NOT sv_bUseProdCounter
         OR (sv_iProdCounterAct = 0 AND sv_iProdCounterRemaining = 0)
         OR (sv_OperationMode < nHalfAutomatic)) THEN

    // Check state of "production limit reached"-alarm
    STATE_ALARM(Name := erProdLimitReached,
            State := State);

    IF State.ALARM_STATE = ALARM_STATE_INACTIVE_ACK THEN
        // Production counter is not used any more
        // or shot counter was reset
        // or production has stopped and alarm is not active any more
        // -> Invalidate event notification
        mbProdEvNotificationActive := FALSE;

        eventNotificationData.dExpirationDate := cUTCZeroDate;
        SET_EVENT(evUpdateEventNotification, eventNotificationData);
        RETURN;
    END_IF;
END_IF;

aCheckAndSendUpdate();

@END_Body

@@@BEG_Comment@@@
@TL(0)

@@@END_Comment@@@

@BEG_Body
@TL(21)
(**************************************** WARNING ********************************************
 *** The KEBA Kemro K2 System including software is not intended for safety control tasks! ***
 ***                       For further information see Comment tab!                        ***
 *********************************************************************************************)

IF mbProdEvNotificationActive AND sv_iProdCounterRemaining = 0 THEN
    // Check state of "production limit reached"-alarm
    STATE_ALARM(Name := erProdLimitReached,
            State := State);

    IF State.ALARM_STATE = ALARM_STATE_INACTIVE_ACK THEN
        // Alarm inactive and quitted
        // -> Invalidate event notification
        mbProdEvNotificationActive := FALSE;
        eventNotificationData.dExpirationDate := cUTCZeroDate;
        SET_EVENT(evUpdateEventNotification, eventNotificationData);
    END_IF;
END_IF;

@END_Body

@@@BEG_Comment@@@
@TL(0)

@@@END_Comment@@@
@END_Body

@END_Contents
